(* CODESYS project tc3_linmot_v1_0_0_3_20150204.library
   Company: NTI AG
   Title: Tc3_LinMot
   Author: NTI AG - LinMot
   Version: 1.0.0.3

Project tree, tasks and I/O mapping:
  libraries: Tc2_Standard, 3.3.0.0 (Beckhoff Automation GmbH)
  Data types/
    internal/
      data type tenLM_AxisState
      data type tstLM_DrvToPlc
      data type tstLM_PlcToDrv
    data type tstLM_Axis
    data type tstLM_CfgCTEntry
    data type tstLM_CfgUPIDListEntry
    data type tstLM_CTEntry
    data type tstLM_LiveParameter
  POUs/
    LinMot Axis Control Function Blocks/
      Unofficial_Unsupported/
        function block LMct_AxisCtrlE12x0_Abort [ST]
      function block LMct_AxisControl [ST]
    LinMot CAM Function Blocks/
      function block LMcm_CAMCtrl [ST]
      function block LMcm_LoadCAM1_mc1100 [ST]
      function block LMcm_LoadCAM1_mc1130 [ST]
      function block LMcm_LoadCAM2_mc1200 [ST]
      function block LMcm_LoadCAM2_mc1230 [ST]
    LinMot Config Function Blocks/
      Unofficial_Unsupported/
        function block LMcf_ParaAccessExt [ST]
      function block LMcf_CTAccess [ST]
      function block LMcf_CurveAccess [ST]
      function block LMcf_GetErrorTxt [ST]
      function block LMcf_GetModUPIDList [ST]
      function block LMcf_ParaAccess [ST]
      function block LMcf_StopStartDefault [ST]
      function block LMcf_WriteUPIDList [ST]
    LinMot Force Control Function Blocks/
      Unofficial_Unsupported/
        function block LMfc_ChangeTargetForceCont [ST]
      function block LMfc_ChangeTargetForce [ST]
      function block LMfc_GoToPosForceCtrlHighLim [ST]
      function block LMfc_GoToPosForceCtrlLowLim [ST]
      function block LMfc_GoToPosRstForceCtrl [ST]
    LinMot Functions/
      function F_GetVersionLinMotLibrary [ST]
      function block LM_F_TRIG [ST]
      function block LM_R_TRIG [ST]
      function LM_UptMCI [ST]
      function USINT_TO_ASCIISTRING [ST]
    LinMot MC Function Blocks/
      Unofficial_Unsupported/
        function block LMmt_IncrTargetPos [ST]
      function block LMmt_GenericMC [ST]
      function block LMmt_IncrActPos [ST]
      function block LMmt_MoveAbs [ST]
      function block LMmt_MoveRel [ST]
      function block LMmt_StartCTCommand [ST]
      function block LMmt_Stop [ST]
      function block LMmt_WriteLivePar [ST]
    LinMot MC Function Blocks Advanced/
      Unofficial_Unsupported/
        function block LMav_PVStreamLREAL [ST]
      function block LMav_CurrentCmdMode [ST]
      function block LMav_Mod16BitCTPar [ST]
      function block LMav_Mod32BitCTPar [ST]
      function block LMav_MoveBestehorn [ST]
      function block LMav_MoveSin [ST]
      function block LMav_PStream [ST]
      function block LMav_PVStream [ST]
      function block LMav_RunCurve [ST]
    Rotary Motors/
      function block LMct_RotaryMotorControl [ST]
      function block LMmt_RotIncrActAngle [ST]
      function block LMmt_RotMoveAbs [ST]
      function block LMmt_RotMoveInfNeg [ST]
      function block LMmt_RotMoveInfPos [ST]
      function block LMmt_RotMoveRel [ST]
  Version/
    global variables Global_Version
  Visualizations/
*)

// Data types/internal/tenLM_AxisState
TYPE tenLM_AxisState :
(*PLC Open like naming of the drive state - ! Has no functionality ! *)
(
	Disabled_LM,
	StandStill_LM,
	Homing_LM,
	ErrorStop_LM,
	Stopping_LM,
	DiscreteMotion_LM,
	ContinuousMotion_LM,
	SynchronizedMotion_LM,
	Jogging_LM
);
END_TYPE

// Data types/internal/tstLM_DrvToPlc
TYPE tstLM_DrvToPlc :
STRUCT
	StateVar 			:UINT; (*StateVar of the drive*)
	StatusWord 			:UINT; (*Statusword of the drive*)
	WarnWord 			:UINT; (*Warnword of the drive*)
	ComActualCurrent16 	:INT; (*16Bit actual current For x11x0 series drive*)
	ComDemandPosition 	:DINT; (*32Bit demand position*)
	ComActualPosition 	:DINT; (*32Bit actual position*)
	ComActualCurrent32 	:DINT; (*32Bit actual current For E1200 series drives*)

	CfgStatusWord 		:UINT; (*Config Channel Status*)
	CfgIndexIn 			:UINT; (*Argument (meaning depends on Cmd ID*)
	CfgValueIn 			:UDINT; (*Argument (meaning depends on Cmd ID*)
END_STRUCT
END_TYPE

// Data types/internal/tstLM_PlcToDrv
TYPE tstLM_PlcToDrv :
STRUCT
	ControlWord 		:UINT; (*ControlWord of the drive*)
	MCHeader 			:UINT; (*Motion command header*)
	MCParaWord0 		:UINT; (*Motion command parameter word 0*)
	MCParaWord1 		:UINT; (*Motion command parameter word 1*)
	MCParaWord2 		:UINT; (*Motion command parameter word 2*)
	MCParaWord3 		:UINT; (*Motion command parameter word 3*)
	MCParaWord4 		:UINT; (*Motion command parameter word 4*)
	MCParaWord5 		:UINT; (*Motion command parameter word 5*)
	MCParaWord6 		:UINT; (*Motion command parameter word 6*)
	MCParaWord7 		:UINT; (*Motion command parameter word 7*)
	MCParaWord8 		:UINT; (*Motion command parameter word 8*)
	MCParaWord9 		:UINT; (*Motion command parameter word 9*)
	MCParaWord10 		:UINT; (*Motion command parameter word 10*)
	MCParaWord11 		:UINT; (*Motion command parameter word 11*)
	MCParaWord12 		:UINT; (*Motion command parameter word 12*)
	MCParaWord13 		:UINT; (*Motion command parameter word 13*)
	MCParaDWord_00_03 	:UDINT; (*Motion command parameter bytes 0-3 (used for E12X0 series drives)*)
	MCParaDWord_04_07 	:UDINT; (*Motion command parameter bytes 4-7 (used for E12X0 series drives)*)
	MCParaDWord_08_11 	:UDINT; (*Motion command parameter bytes 8-11 (used for E12X0 series drives)*)
	MCParaDWord_12_15 	:UDINT; (*Motion command parameter bytes 12-15 (used for E12X0 series drives)*)
	MCParaDWord_16_19 	:UDINT; (*Motion command parameter bytes 16-19 (used for E12X0 series drives)*)
	MCParaDWord_20_23 	:UDINT; (*Motion command parameter bytes 20-23 (used for E12X0 series drives)*)
	MCParaDWord_24_27 	:UDINT; (*Motion command parameter bytes 24-27 (used for E12X0 series drives)*)

	CfgControlWord 		:UINT; (*Config Channel Control*)
	CfgIndexOut 		:UINT; (*Argument (meaning depends on Cmd ID*)
	CfgValueOut 		:UDINT; (*Argument (meaning depends on Cmd ID*)
END_STRUCT
END_TYPE

// Data types/tstLM_Axis
TYPE tstLM_Axis : 
STRUCT
	PlcToDrv			AT%Q* :tstLM_PlcToDrv; (*PLC to Drive struct*)
	DrvToPlc			AT%I* :tstLM_DrvToPlc; (*Drive to PLC struct*)
	(*Status information*)
	AxisState			:tenLM_AxisState;
	CommandRunning		:BOOL;
	CommandAborted		:BOOL;
	ConfigChannelBusy	:BOOL;
	(*Information (Not required for prober work of the library function blocks)*)
	AxisName			:STRING;
	AxisNr				:UINT;
	AxisCtrlType		:STRING; (*Eg. 'E1200-EC-UC', 'E1130-DP', 'B1100-GP', ....*)
END_STRUCT
END_TYPE

// Data types/tstLM_CfgCTEntry
TYPE tstLM_CfgCTEntry :
STRUCT
	CTID		:UINT; (*ID of command table entry*)
	BlockSize	:UINT; (*Size of EntryBlock in Bytes*)
	DataBlock	:ARRAY[0..15] OF UDINT; (*EntryBlock, 64Bytes*)

(*Example of a Command Table Entry Data Block:
0002A701h, 	LowWord = Entry Version ID (fix A701h) / HighWord = Sequenced Entry ID
00000100h,	LowWord: Motion Cmd Header(010xh=VAI Go To Pos) / HighWord: Motion Cmd Par Byte 0..1
42400000h, 	Motion Cmd Par Byte 2..5
4240000Fh, 	Motion Cmd Par Byte 6..9
4240000Fh, 	Motion Cmd Par Byte 10..13
0000000Fh, 	Motion Cmd Par Byte 14..17
00000000h, 	Motion Cmd Par Byte 18..21
00000000h, 	Motion Cmd Par Byte 22..25
00000000h, 	Motion Cmd Par Byte 26..29
6E550000h, 	LowWord: Motion Cmd Par Byte 30..31 / HighWord: Entry Name Character 0..1
656D616Eh, 	Entry Name Character 2..5
00000064h, 	Entry Name Character 6..9
00000000h, 	Entry Name Character 10..13
FFFF0000h, 	LowWord: Entry Name Character 14..15 / HighWord: Reserved for future use
FFFFFFFFh, 	Reserved for future use
FFFFFFFFh, 	Reserved for future use
*)
END_STRUCT
END_TYPE

// Data types/tstLM_CfgUPIDListEntry
TYPE tstLM_CfgUPIDListEntry :
STRUCT
	UPID		:UINT; (*LinMot parameter, UPID [Unique Parameter ID]*)
	UPIDValue	:UDINT; (*Value of the parameter*)
END_STRUCT
END_TYPE

// Data types/tstLM_CTEntry
TYPE tstLM_CTEntry :
STRUCT
	CTEntryID	:INT;
	ParaOffset	:INT;
	ParaValue	:DINT;
END_STRUCT
END_TYPE

// Data types/tstLM_LiveParameter
TYPE tstLM_LiveParameter :
STRUCT
	UPID		:UINT;
	UPIDValue	:DINT;
END_STRUCT
END_TYPE

// Version/Global_Version
// This function has been automatically generated from the project information.
VAR_GLOBAL CONSTANT
	{attribute 'const_non_replaced'}
	stLibVersion_Tc3_LinMot : ST_LibVersion := (iMajor := 1, iMinor := 0, iBuild := 0, iRevision := 3, sVersion := '1.0.0.3');
END_VAR

// POUs/LinMot Axis Control Function Blocks/Unofficial_Unsupported/LMct_AxisCtrlE12x0_Abort
FUNCTION_BLOCK LMct_AxisCtrlE12x0_Abort
VAR_INPUT
	SwitchOn			:BOOL;	(*Switch on motor*)
	Abort_INV			:BOOL;	(*/Abort*)
	Home				:BOOL;	(*Start homing procedure*)
	ErrorAcknowledge	:BOOL;	(*Error acknowledge*)
	JogPlus				:BOOL;	(*Jog move postive*)
	JogMinus			:BOOL;	(*Jog move negative*)
END_VAR
VAR_IN_OUT
	Axis				:tstLM_Axis; (*Axis reference*)
END_VAR
VAR_OUTPUT
	OperationEnabled	:BOOL;	(*Axis powered on*)
	Aborting			:BOOL;	(*Aborting*)
	SwitchOnLocked		:BOOL;	(*Switch on locked*)
	Homed				:BOOL;	(*Axis has reference*)
	MotionActive		:BOOL;	(*Motion active (Setpoint generation (VAI, curve) active)*)
	Jogging				:BOOL;	(*Axis is moving in jog mode*)
	Warning				:BOOL;	(*Warning detected*)
	Error				:BOOL; 	(*Error detected*)
	ErrorCode			:UINT;	(*Error code, see MotionCtrlSW manual*)
	ActualPosition		:REAL;	(*Actual position in [mm]*)
	ActualCurrent		:REAL;	(*Actual motor current in [A]*)
END_VAR
VAR
	uiState				:UINT;	(*internal -> Current state of the drive*)
	rTrigHome 			:LM_R_TRIG;	(*internal ->*)
	rTrigHomed 			:LM_R_TRIG;	(*internal ->*)
	bRehome 			:BOOL; 	(*internal ->*)
END_VAR
(*Version history:
Date         	 | Version    	| Created under     		| Author          		| Remark 
------------------------------------------------------------------------------------------------------------------------------- 
2011-jul-12   	 | 1.0.0      	| V2.11.0 (Build 1016)		| fj  					| initial release 
2011-nov-22   	 | 1.0.1      	| V2.11.0 (Build 1016)		| fj  					| homed output reset if home input is set 
2011-dec-01   	 | 1.0.2      	| V2.11.0 (Build 1016)		| fj  					| code optimisation
2012-jan-25   	 | 1.0.3     	| V2.11.0 (Build 1016)		| fj  					| operation enabled output is now directly mapped to the status word bit 0
2012-may-01  	 | 1.1.0b     	| V2.11.0 (Build 1016)		| fj  					| added /Abort input
2012-aug-21  	 | 1.1.0c     	| V2.11.0 (Build 1016)		| fj  					| added additional StateVar check for 090Fh ("homing finished") when rehoming
*)

(*Eingänge zuweisen/lesen ][ Read and allocate inputs*)
	ActualPosition := DINT_TO_REAL(Axis.DrvToPlc.ComActualPosition)/10000;
    	ActualCurrent := DINT_TO_REAL(Axis.DrvToPlc.ComActualCurrent32)/1000;

(*Variablen ][ variables*)
	uiState := SHR(Axis.DrvToPlc.StateVar, 8);
	SwitchOnLocked := Axis.DrvToPlc.StatusWord.6;
	Warning := Axis.DrvToPlc.StatusWord.7;
	Homed := Axis.DrvToPlc.StatusWord.11;
	MotionActive := Axis.DrvToPlc.StatusWord.13;
	OperationEnabled	:= Axis.DrvToPlc.StatusWord.0;

(*	IF uiState = 16#08 THEN
		OperationEnabled	:= Axis.DrvToPlc.StatusWord.0;
	ELSE
		OperationEnabled	:= FALSE;
	END_IF
*) (*Disabled 2012/01/25 fj*)
(*=============================================================================
*  State Machine
===============================================================================*)    

CASE uiState OF
	(*Not Ready to Switch On*)
	00:	Axis.AxisState := Disabled_LM;

	(*State 4: Error*)
	04:	ErrorCode := UINT_TO_USINT(Axis.DrvToPlc.StateVar);
           	Error := TRUE;
		Axis.AxisState := ErrorStop_LM;

	(*State 8: Operation Enabled*)
	08:	Homed := Axis.DrvToPlc.StateVar.7;
		IF Axis.DrvToPlc.StatusWord.13 AND NOT (Axis.AxisState = Stopping_LM) THEN
			Axis.AxisState := DiscreteMotion_LM;
		ELSIF NOT Axis.DrvToPlc.StatusWord.13 AND NOT (Axis.AxisState = Stopping_LM) THEN
			Axis.AxisState := StandStill_LM;
		END_IF

	(*State 9: Homing*)
	09:	Axis.AxisState := Homing_LM;

	(*State 12: Aborting*)
	12:	Aborting := TRUE;
		IF Axis.DrvToPlc.StatusWord.13 THEN
			Axis.AxisState := Stopping_LM;
		ELSE
			Axis.AxisState := StandStill_LM;
		END_IF

	(*State 14: Error Behaviour QuickStop*)
	14:	Axis.AxisState := ErrorStop_LM;

	(*State 16: Jogging +*)
	16:	Axis.AxisState := Jogging_LM;

	(*State 17: Jogging -*)
	17:	Axis.AxisState := Jogging_LM;

END_CASE;


(*Wenn der drive nicht im Fehlerzustand ist, werden Error und ErrorCode auf Null gesetzt*)
(*If the drive is not in Error state, Error and ErrorCode are set to zero*)
IF uiState <> 16#04 THEN
        	Error := FALSE;
        	ErrorCode := 16#00;
END_IF;

IF uiState <> 16#08 THEN
        	Axis.PlcToDrv.MCHeader := 16#0000; (*Reset Header to prevent "MC Cmd in wrong state" error*)
	Axis.CommandRunning := FALSE;
	Axis.CommandAborted := FALSE;
END_IF;

(*Switch On*)
Axis.PlcToDrv.ControlWord.0 := SwitchOn;
IF NOT Axis.PlcToDrv.ControlWord.0 AND NOT (uiState = 4 OR uiState = 12 OR uiState = 14) THEN
	Axis.AxisState := Disabled_LM;
END_IF

(*Home*)
Axis.PlcToDrv.ControlWord.11 := Home;
rTrigHome(CLK:=Home);
rTrigHomed(CLK:=Axis.DrvToPlc.StatusWord.11);

IF rTrigHome.Q AND (uiState = 8) THEN
	bRehome := TRUE;
END_IF
IF bRehome THEN
	Homed := FALSE;
	IF rTrigHomed.Q OR (Axis.DrvToPlc.StateVar = 16#090F) THEN
 		bRehome := FALSE;
  		Homed := Axis.DrvToPlc.StatusWord.11;
	END_IF
END_IF

(*Error acknowledge*)
Axis.PlcToDrv.ControlWord.7 := ErrorAcknowledge;

(*JogPlus*)
Axis.PlcToDrv.ControlWord.8 := JogPlus;

(*JogMinus*)
Axis.PlcToDrv.ControlWord.9 := JogMinus;

IF (uiState = 16 OR uiState = 17) AND UINT_TO_USINT(Axis.DrvToPlc.StateVar) = 16#01 THEN
	Jogging := TRUE;
ELSE
	Jogging := FALSE;
END_IF

(*/Abort*)
Axis.PlcToDrv.ControlWord.4 := Abort_INV;
IF NOT Abort_INV THEN
	Axis.CommandAborted := TRUE;
ELSE
	Aborting := FALSE;
END_IF

END_FUNCTION_BLOCK

// POUs/LinMot Functions/LM_R_TRIG
FUNCTION_BLOCK LM_R_TRIG
(* Rising Edge detection *)
VAR_INPUT
	CLK	:BOOL;	(*Signal to detect*)
END_VAR
VAR_OUTPUT
	Q	:BOOL;	(*Edge detected*)
END_VAR
VAR
	M	:BOOL;
END_VAR
(*Version history:
Date         	 | Version    		| Created under     	| Author          	| Remark 
------------------------------------------------------------------------------------------------------------------------------- 
2013-nov-27   	 | 1.0.0      		| V2.11.0 (Build 1016)	| fj  				| initial release 
*)

(*Bildung der positiven Flanke  // get the positive pulse*)
    Q  := CLK AND NOT M;
    M  := CLK;

END_FUNCTION_BLOCK

// POUs/LinMot Axis Control Function Blocks/LMct_AxisControl
FUNCTION_BLOCK LMct_AxisControl
VAR_INPUT
	SwitchOn		    :BOOL;	(*Switch on motor*)
	Home				:BOOL;	(*Start homing procedure*)
	ErrorAcknowledge	:BOOL;	(*Error acknowledge*)
	JogPlus				:BOOL;	(*Jog move postive*)
	JogMinus			:BOOL;	(*Jog move negative*)
END_VAR
VAR_IN_OUT
	Axis	       		:tstLM_Axis; (*Axis reference*)
END_VAR
VAR_OUTPUT
	OperationEnabled	:BOOL;	(*Axis powered on*)
	SwitchOnLocked		:BOOL;	(*Switch on locked*)
	Homed     	      	:BOOL;	(*Axis has reference*)
	MotionActive		:BOOL;	(*Motion active (Setpoint generation (VAI, curve) active)*)
	Jogging				:BOOL;	(*Axis is moving in jog mode*)
	Warning         	:BOOL;	(*Warning detected*)
	Error          		:BOOL;	(*Error detected*)
	ErrorCode      		:UINT;	(*Error code, see MotionCtrlSW manual*)
	DemandPosition  	:REAL;	(*Demand position in [mm]*)
	ActualPosition  	:REAL;	(*Actual position in [mm]*)
	ActualCurrent   	:REAL;	(*Actual motor current in [A]*)
END_VAR
VAR
	uiState        		:UINT;	(*internal -> Current state of the drive*)
	rTrigHome 			:LM_R_TRIG;	(*internal ->*)
	fTrigHome 			:LM_F_TRIG;	(*internal ->*)
END_VAR
(*Version history:
Date         	 | Version    		| Created under     	| Author          	| Remark 
------------------------------------------------------------------------------------------------------------------------------- 
2011-jul-12   	 | 1.0.0      		| V2.11.0 (Build 1016)	| fj  				| initial release 
2011-nov-22   	 | 1.0.1      		| V2.11.0 (Build 1016)	| fj  				| homed output reset if home input is set 
2011-dec-01   	 | 1.0.2      		| V2.11.0 (Build 1016)	| fj  				| code optimisation
2012-jan-25   	 | 1.0.3     		| V2.11.0 (Build 1016)	| fj  				| operation enabled output is now directly mapped to the status word bit 0
2012-oct-16   	 | 1.1.0      		| V2.11.0 (Build 1016)	| fj  				| added additional StateVar check for 090Fh ("homing finished") when rehoming
2014-may-13   	 | 1.0.0.1     		| v3.14014.0			| fj  				| added output DemandPosition
																				| optimized home input / homed output behaviour
*)

(*Eingänge zuweisen/lesen ][ Read and allocate inputs*)
	ActualPosition := DINT_TO_REAL(Axis.DrvToPlc.ComActualPosition)/10000;
	DemandPosition := DINT_TO_REAL(Axis.DrvToPlc.ComDemandPosition)/10000;
	(*Workaround for different XML current definitions (16Bit/32Bit)*)
	IF Axis.DrvToPlc.ComActualCurrent32 = 0 AND Axis.DrvToPlc.ComActualCurrent16 = 0 THEN
		ActualCurrent := 0;
	ELSIF Axis.DrvToPlc.ComActualCurrent32 <> 0 AND Axis.DrvToPlc.ComActualCurrent16 = 0 THEN
		ActualCurrent := DINT_TO_REAL(Axis.DrvToPlc.ComActualCurrent32)/1000;
	ELSIF Axis.DrvToPlc.ComActualCurrent32 = 0 AND Axis.DrvToPlc.ComActualCurrent16 <> 0 THEN
		ActualCurrent := INT_TO_REAL(Axis.DrvToPlc.ComActualCurrent16)/1000;
	ELSE
		ActualCurrent := DINT_TO_REAL(Axis.DrvToPlc.ComActualCurrent32)/1000; (*If both 16/32Bit currents aren't 0 32Bit has higher priority*)
	END_IF

(*Variablen ][ variables*)
	uiState := SHR(Axis.DrvToPlc.StateVar, 8);
	SwitchOnLocked := Axis.DrvToPlc.StatusWord.6;
	Warning := Axis.DrvToPlc.StatusWord.7;
	MotionActive := Axis.DrvToPlc.StatusWord.13;
	OperationEnabled := Axis.DrvToPlc.StatusWord.0;

(*=============================================================================
*  State Machine
===============================================================================*)    

CASE uiState OF
	(*Not Ready to Switch On*)
	00:	Axis.AxisState := Disabled_LM;

	(*State 4: Error*)
	04:	ErrorCode := UINT_TO_USINT(Axis.DrvToPlc.StateVar);
		Error := TRUE;
		Axis.AxisState := ErrorStop_LM;

	(*State 8: Operation Enabled*)
	08:	Homed := Axis.DrvToPlc.StateVar.7;
		IF Axis.DrvToPlc.StatusWord.13 AND NOT (Axis.AxisState = Stopping_LM) THEN
			Axis.AxisState := DiscreteMotion_LM;
		ELSIF NOT Axis.DrvToPlc.StatusWord.13 AND NOT (Axis.AxisState = Stopping_LM) THEN
			Axis.AxisState := StandStill_LM;
		END_IF

	(*State 9: Homing*)
	09:	Axis.AxisState := Homing_LM;
		IF Axis.DrvToPlc.StateVar = 16#090F THEN
			Axis.PlcToDrv.ControlWord.11 := FALSE;
		END_IF

	(*State 14: Error Behaviour QuickStop*)
	14:	Axis.AxisState := ErrorStop_LM;

	(*State 16: Jogging +*)
	16:	Axis.AxisState := Jogging_LM;

	(*State 17: Jogging -*)
	17:	Axis.AxisState := Jogging_LM;

END_CASE;


(*Wenn der drive nicht im Fehlerzustand ist, werden Error und ErrorCode auf Null gesetzt*)
(*If the drive is not in Error state, Error and ErrorCode are set to zero*)
IF uiState <> 16#04 THEN
	Error := FALSE;
	ErrorCode := 16#00;
END_IF;

IF uiState <> 16#08 THEN
	Axis.PlcToDrv.MCHeader := 16#0000; (*Reset Header to prevent "MC Cmd in wrong state" error*)
	Axis.CommandRunning := FALSE;
	Axis.CommandAborted := FALSE;
END_IF;

(*Switch On*)
Axis.PlcToDrv.ControlWord.0 := SwitchOn;
IF NOT Axis.PlcToDrv.ControlWord.0 AND NOT (uiState = 4 OR uiState = 14) THEN
	Axis.AxisState := Disabled_LM;
END_IF

(*Home*)
rTrigHome(CLK:=Home);
fTrigHome(CLK:=Home);
IF rTrigHome.Q THEN
	Axis.PlcToDrv.ControlWord.11 := TRUE;
END_IF
IF fTrigHome.Q  THEN
	Axis.PlcToDrv.ControlWord.11 := FALSE;
END_IF

IF uiState = 16#09 OR (Axis.PlcToDrv.ControlWord.11 AND NOT (uistate = 16#09)) THEN
	Homed := FALSE;
ELSE
	Homed := Axis.DrvToPlc.StatusWord.11;
END_IF

(*Error acknowledge*)
Axis.PlcToDrv.ControlWord.7 := ErrorAcknowledge;

(*JogPlus*)
Axis.PlcToDrv.ControlWord.8 := JogPlus;

(*JogMinus*)
Axis.PlcToDrv.ControlWord.9 := JogMinus;

IF (uiState = 16 OR uiState = 17) AND UINT_TO_USINT(Axis.DrvToPlc.StateVar) = 16#01 THEN
	Jogging := TRUE;
ELSE
	Jogging := FALSE;
END_IF

END_FUNCTION_BLOCK

// POUs/LinMot Functions/LM_F_TRIG
FUNCTION_BLOCK LM_F_TRIG
(* Falling Edge detection *)
VAR_INPUT
	CLK	:BOOL;	(*Signal to detect*)
END_VAR
VAR_OUTPUT
	Q	:BOOL;	(*Edge detected*)
END_VAR
VAR
	M	:BOOL;
END_VAR
(*Version history:
Date         	 | Version    		| Created under     	| Author          	| Remark 
------------------------------------------------------------------------------------------------------------------------------- 
2013-nov-27   	 | 1.0.0      		| V2.11.0 (Build 1016)	| fj  				| initial release 
*)

(*Bildung der negativen Flanke  // get the negative pulse*)
    Q  := NOT CLK AND M;
    M  := CLK;

END_FUNCTION_BLOCK

// POUs/LinMot CAM Function Blocks/LMcm_CAMCtrl
FUNCTION_BLOCK LMcm_CAMCtrl
VAR_INPUT
	Execute			:BOOL;	(*Execute command*)
	Mode			:UINT;	(*Mode 0: CAM Enable
 							Mode 1: CAM Disable
 							Mode 2: CAM Go To Sync Pos
 							Mode 3: Encoder CAM Set Value [Inputs used: EncValue]
							Mode 4: Encoder CAM 1 Enable
							Mode 5: Encoder CAM 1 Disable
							Mode 6: Encoder CAM 2 Enable
							Mode 7: Encoder CAM 2 Disable
							*)
	EncValue		:UDINT;	(*Encoder value to be written*)
END_VAR
VAR_IN_OUT
	Axis	        			:tstLM_Axis; (*Axis reference*)
END_VAR
VAR_OUTPUT
	Done			:BOOL;	(*Command has been executed*)
	Busy			:BOOL;	(*Command running / FB Busy*)
	Error          	:BOOL;	(*Error detected*)
	ErrorID 		:UINT;	(*Error ID:
							01h: Axis not ready
 							02h: Axis already has command running
 							03h: Axis has error
 							04h: Command interrupted
 							05h: Command aborted
							06h: Invalid input(s)
							*)
END_VAR
VAR
	usiOldCmdCount 	:USINT;	(*internal -> *)
	usiNewCmdCount	:USINT; 	(*internal -> *)
	uiCState		:UINT;     	(*internal -> *)
	uiFbState		:UINT;	(*internal -> *)
	rTrig			:LM_R_TRIG;	(*internal -> *)
	uiCmdHeader		:UINT;	(*internal -> *)
END_VAR

(*Version history:
Date         	 | Version    		| Created under     	| Author       		| Remark 
------------------------------------------------------------------------------------------------------------------------------- 
2012-aug-30   	 | 1.1.0     		| V2.11.0 (Build 1016)	| fj  				| initial release
2013-nov-27   	 | 1.1.1      		| V2.11.0 (Build 1016)	| fj  				| check if command done fixed
*)

	usiOldCmdCount := SHR(UINT_TO_USINT(SHL(Axis.DrvToPlc.StateVar,4)),4);
	uiCState := SHR(Axis.DrvToPlc.StateVar, 8);

(*Flankenerkennung am Execute Eingang*)
(*Edge detection on Execute input*)
rTrig(CLK:=Execute);
IF rTrig.Q AND Mode = 2 AND uiCState = 16#08 AND Axis.DrvToPlc.StateVar.6 AND NOT Axis.CommandRunning THEN (*Start command if mode = 2*)
	Axis.CommandRunning := TRUE;
	Busy := TRUE;
	uiFbState := 1;
ELSIF rTrig.Q AND Mode <> 2 AND NOT  Axis.CommandRunning THEN (*Start command if mode <> 2*)
	Axis.CommandRunning := TRUE;
	Busy := TRUE;
	uiFbState := 1;
ELSIF rTrig.Q AND Mode = 2 AND (uiCState <> 16#08 OR NOT Axis.DrvToPlc.StateVar.6) THEN (*Axis not ready*)
	uiFbState := 50; (*Error state*)
	Error := TRUE;
	ErrorID := 16#01; (*Axis not ready*)
ELSIF rTrig.Q AND Axis.CommandRunning AND NOT Busy THEN (*Axis already has a command running*)
	uiFbState := 50; (*Error state*)
	Error := TRUE;
	ErrorID := 16#02; (*Axis already has a command running*)
END_IF

IF Busy AND Mode = 2 AND uiCState = 16#04 THEN
	Axis.CommandRunning := FALSE;
	uiFbState := 50;
	Error := TRUE;
	ErrorID := 16#03; (*Axis has error*)
END_IF

IF Busy AND Mode = 2 AND uiCState <> 16#08 THEN
	Axis.CommandRunning := FALSE;
	uiFbState := 50; (*Error state*)
	Error := TRUE;
	ErrorID := 16#04; (*Command interupted*)
ELSIF Busy AND Axis.CommandAborted THEN
	uiFbState := 50; (*Error state*)
	Error := TRUE;
	ErrorID := 16#05; (*Command aborted*)
END_IF

(*State machine*)
CASE uiFbState OF
	0:	;

	1:     	(*Befehlskopf mit CMD Count berechen und senden ][ Calculate and send command header*)
		CASE Mode OF
			0:	uiCmdHeader := 16#1000; (*CAM Enable*)
			1:	uiCmdHeader := 16#1010; (*CAM Disable*)
			2:	uiCmdHeader := 16#1020; (*CAM Go To Sync Pos*)
			3:	uiCmdHeader := 16#1040; (*Encoder CAM Set Value*)
			4:	uiCmdHeader := 16#1160; (*Encoder CAM 1 Enable*)
			5:	uiCmdHeader := 16#1170; (*Encoder CAM 1 Disable*)
			6:	uiCmdHeader := 16#1260; (*Encoder CAM 2 Enable*)
			7:	uiCmdHeader := 16#1270; (*Encoder CAM 2 Disable*)
		END_CASE

		usiNewCmdCount := (usiOldCmdCount + 1) MOD 16 ; (*MOD 16*)
     	   	Axis.PlcToDrv.MCHeader := 16#0000; (*Reset Header*)
     	   	Axis.PlcToDrv.MCHeader := uiCmdHeader + usiNewCmdCount;

		IF Mode = 3 THEN
			Axis.PlcToDrv.MCParaWord0 := UDINT_TO_UINT(EncValue);
			Axis.PlcToDrv.MCParaWord1 := UDINT_TO_UINT(ROR(EncValue,16));
		ELSE
			Axis.PlcToDrv.MCParaWord0 := 0;
			Axis.PlcToDrv.MCParaWord1 := 0;
		END_IF

		LM_UptMCI(Axis);

		uiFbState := 2;

	2:	(*Prüfen ob Befehl ausgeführt ][ Check if command has been executed*)
		IF (Mode = 2 AND (usiOldCmdCount = usiNewCmdCount) AND uiCState = 16#08 AND Axis.DrvToPlc.StateVar.6)
			OR ((Mode <> 2) AND (usiOldCmdCount = usiNewCmdCount)) THEN
			Done := TRUE;
			Busy := FALSE;
	     	   	Axis.PlcToDrv.MCHeader := 16#0000 + usiNewCmdCount; (*Send no operation*)
			Axis.CommandRunning := FALSE;
			uiFbState := 3;
		END_IF

	3:	IF NOT Execute THEN
			uiFbState := 0;
			Busy := FALSE;
			Done := FALSE;
		END_IF

	50:	Error := TRUE;
		Busy := FALSE;
		Done := FALSE;
		IF NOT Execute THEN
			uiFbState := 0;
			Error := FALSE;
			ErrorID := 0;
		END_IF

END_CASE

END_FUNCTION_BLOCK

// POUs/LinMot Functions/LM_UptMCI
FUNCTION LM_UptMCI : bool
VAR_IN_OUT
	Axis 	:tstLM_Axis;
END_VAR
VAR
END_VAR

Axis.PlcToDrv.MCParaDWord_00_03 := SHL(UINT_TO_UDINT(Axis.PlcToDrv.MCParaWord1),16) + UINT_TO_UDINT(Axis.PlcToDrv.MCParaWord0);
Axis.PlcToDrv.MCParaDWord_04_07 := SHL(UINT_TO_UDINT(Axis.PlcToDrv.MCParaWord3),16) + UINT_TO_UDINT(Axis.PlcToDrv.MCParaWord2);
Axis.PlcToDrv.MCParaDWord_08_11 := SHL(UINT_TO_UDINT(Axis.PlcToDrv.MCParaWord5),16) + UINT_TO_UDINT(Axis.PlcToDrv.MCParaWord4);
Axis.PlcToDrv.MCParaDWord_12_15 := SHL(UINT_TO_UDINT(Axis.PlcToDrv.MCParaWord7),16) + UINT_TO_UDINT(Axis.PlcToDrv.MCParaWord6);
Axis.PlcToDrv.MCParaDWord_16_19 := SHL(UINT_TO_UDINT(Axis.PlcToDrv.MCParaWord9),16) + UINT_TO_UDINT(Axis.PlcToDrv.MCParaWord8);
Axis.PlcToDrv.MCParaDWord_20_23 := SHL(UINT_TO_UDINT(Axis.PlcToDrv.MCParaWord11),16) + UINT_TO_UDINT(Axis.PlcToDrv.MCParaWord10);
Axis.PlcToDrv.MCParaDWord_24_27 := SHL(UINT_TO_UDINT(Axis.PlcToDrv.MCParaWord13),16) + UINT_TO_UDINT(Axis.PlcToDrv.MCParaWord12);

END_FUNCTION

// POUs/LinMot CAM Function Blocks/LMcm_LoadCAM1_mc1100
FUNCTION_BLOCK LMcm_LoadCAM1_mc1100
VAR_INPUT
	Execute			:BOOL;    	(*Execute Command*)
	CurveID			:UINT;     	(*Curve ID*)
	CurveStartCount	:UDINT;	(*Curve Start Count [Incr]*)
END_VAR
VAR_IN_OUT
	Axis			:tstLM_Axis; (*Axis struct*)
END_VAR
VAR_OUTPUT
	Done			:BOOL;	(*Command has been executed*)
	Busy			:BOOL;	(*Command running / FB Busy*)
	Error			:BOOL;	(*Error detected*)
	ErrorID			:UINT;	(*Error ID:
							01h: Axis not ready
 							02h: Axis already has command running
 							03h: Axis has error
 							04h: Command interrupted
 							05h: Command aborted
							06h: Invalid input(s)
							*)
END_VAR
VAR
	usiOldCmdCount 	:USINT;	(*internal -> *)
	usiNewCmdCount	:USINT;	(*internal -> *)
	uiCState		:UINT;	(*internal -> *)
	uiFbState		:UINT;	(*internal -> *)
	rTrig			:LM_R_TRIG;	(*internal -> *)
	udiTmpDWord		:UDINT;	(*internal -> *)

 	uiCmdHeader 	:UINT := 16#1100;	(*CommandHeader (110xh) of the "Encoder CAM 1 Define Curve With Default Parameters (110xh)" motion command*)
END_VAR
(*Version history:
Date         	 | Version    	| Created under     		| Author          		| Remark 
------------------------------------------------------------------------------------------------------------------------------- 
2012-aug-30   	 | 1.1.0     		| V2.11.0 (Build 1016)	| fj  				| initial release
*)

(*Variablen ][ variables*)
	usiOldCmdCount := SHR(UINT_TO_USINT(SHL(Axis.DrvToPlc.StateVar,4)),4);
	uiCState := SHR(Axis.DrvToPlc.StateVar, 8);

(*Flankenerkennung am Execute Eingang*)
(*Edge detection on Execute input*)
rTrig(CLK:=Execute);
IF rTrig.Q AND uiCState = 16#08 AND NOT Axis.CommandRunning THEN (*Start command*)
	Axis.CommandRunning := TRUE;
	Busy := TRUE;
	uiFbState := 1;
ELSIF rTrig.Q AND Busy THEN (*Restart command / New rising edge on execute input*)
	Axis.CommandRunning := TRUE;
	Busy := TRUE;
	uiFbState := 1;
ELSIF rTrig.Q AND uiCState <> 16#08 THEN (*Axis not ready*)
	uiFbState := 50; (*Error state*)
	Error := TRUE;
	ErrorID := 16#01; (*Axis not ready*)
ELSIF rTrig.Q AND Axis.CommandRunning AND NOT Busy THEN (*Axis already has a command running*)
	uiFbState := 50; (*Error state*)
	Error := TRUE;
	ErrorID := 16#02; (*Axis already has a command running*)
END_IF

IF Busy AND uiCState = 16#04 THEN
	Axis.CommandRunning := FALSE;
	uiFbState := 50;
	Error := TRUE;
	ErrorID := 16#03; (*Axis has error*)
END_IF

IF Busy AND uiCState <> 16#08 THEN
	Axis.CommandRunning := FALSE;
	uiFbState := 50; (*Error state*)
	Error := TRUE;
	ErrorID := 16#04; (*Command interupted*)
ELSIF Busy AND Axis.CommandAborted THEN
	uiFbState := 50; (*Error state*)
	Error := TRUE;
	ErrorID := 16#05; (*Command aborted*)
END_IF

(*State machine*)
CASE uiFbState OF
	0:	;

	1:	IF (1 <= CurveID AND CurveID <= 100)
		AND (0 <= CurveStartCount AND CurveStartCount <= 4294967295)
		THEN
			(*Befehlskopf mit CMD Count berechen und senden ][ Calculate and send command header*)
			usiNewCmdCount := (usiOldCmdCount + 1) MOD 16 ; (*MOD 16*)
			Axis.PlcToDrv.MCHeader := 16#0000; (*Reset Header*)
			Axis.PlcToDrv.MCHeader := uiCmdHeader + usiNewCmdCount;
	
			Axis.PlcToDrv.MCParaWord0 := CurveID; (*Curve ID*)
	
			Axis.PlcToDrv.MCParaWord1 := UDINT_TO_UINT(CurveStartCount); (*Curve Start Count*)
			Axis.PlcToDrv.MCParaWord2 := UDINT_TO_UINT(ROR(CurveStartCount,16));

			LM_UptMCI(Axis);

			uiFbState := 2;
		ELSE
			Axis.CommandRunning := FALSE;
			uiFbState := 50; (*Error state*)
			Error := TRUE;
			ErrorID := 16#06; (*Invalid input(s)*)
		END_IF

	2:	(*Prüfen ob Befehl ausgeführt ][ Check if command has been executed*)
		IF usiOldCmdCount = usiNewCmdCount AND uiCState = 16#08 THEN
			Done := TRUE;
			Busy := FALSE;
			Axis.PlcToDrv.MCHeader := 16#0000 + usiNewCmdCount; (*Send no operation*)
			Axis.CommandRunning := FALSE;
			uiFbState := 3;
		END_IF

	3:	IF NOT Execute THEN
			uiFbState := 0;
			Busy := FALSE;
			Done := FALSE;
		END_IF

	50:	Error := TRUE;
		Busy := FALSE;
		Done := FALSE;
		IF NOT Execute THEN
			uiFbState := 0;
			Error := FALSE;
			ErrorID := 0;
		END_IF

END_CASE

END_FUNCTION_BLOCK

// POUs/LinMot CAM Function Blocks/LMcm_LoadCAM1_mc1130
FUNCTION_BLOCK LMcm_LoadCAM1_mc1130
VAR_INPUT
	Execute			:BOOL;	(*Execute Command*)
	CurveID			:UINT;	(*Curve ID*)
	CurveStartCount	:UDINT;	(*Curve Start Count [Incr]*)
	OffsetPosition	:REAL;	(*Offset Position [mm]*)
	TargetPosition	:REAL;	(*Target Positon [mm]*)
	CurveLength		:UDINT;	(*Curve Length [Incr]*)
END_VAR
VAR_IN_OUT
	Axis			:tstLM_Axis; (*Axis struct*)
END_VAR
VAR_OUTPUT
	Done			:BOOL;	(*Command has been executed*)
	Busy			:BOOL;	(*Command running / FB Busy*)
	Error			:BOOL;	(*Error detected*)
	ErrorID			:UINT;	(*Error ID:
							01h: Axis not ready
 							02h: Axis already has command running
 							03h: Axis has error
 							04h: Command interrupted
 							05h: Command aborted
							06h: Invalid input(s)
							*)
END_VAR
VAR
	usiOldCmdCount 	:USINT;	(*internal -> *)
	usiNewCmdCount	:USINT;	(*internal -> *)
	uiCState		:UINT;	(*internal -> *)
	uiFbState		:UINT;	(*internal -> *)
	rTrig			:LM_R_TRIG;	(*internal -> *)
	udiTmpDWord		:UDINT;	(*internal -> *)

 	uiCmdHeader 	:UINT := 16#1130;	(*CommandHeader (113xh) of the "Encoder CAM 1 Define Curve From Pos To Pos In Counts (113xh)" motion command*)
END_VAR
(*Version history:
Date         	 | Version    	| Created under     		| Author          		| Remark 
------------------------------------------------------------------------------------------------------------------------------- 
2011-jul-12   	 | 1.0.0      		| V2.11.0 (Build 1016)	| fj  				| initial release 
2011-dec-01   	 | 1.0.2      		| V2.11.0 (Build 1016)	| fj  				| code optimisation
2012-apr-25   	 | 1.1.0     		| V2.11.0 (Build 1016)	| fj  				| added input parameters check
*)

(*Variablen ][ variables*)
	usiOldCmdCount := SHR(UINT_TO_USINT(SHL(Axis.DrvToPlc.StateVar,4)),4);
	uiCState := SHR(Axis.DrvToPlc.StateVar, 8);

(*Flankenerkennung am Execute Eingang*)
(*Edge detection on Execute input*)
rTrig(CLK:=Execute);
IF rTrig.Q AND uiCState = 16#08 AND NOT Axis.CommandRunning THEN (*Start command*)
	Axis.CommandRunning := TRUE;
	Busy := TRUE;
	uiFbState := 1;
ELSIF rTrig.Q AND Busy THEN (*Restart command / New rising edge on execute input*)
	Axis.CommandRunning := TRUE;
	Busy := TRUE;
	uiFbState := 1;
ELSIF rTrig.Q AND uiCState <> 16#08 THEN (*Axis not ready*)
	uiFbState := 50; (*Error state*)
	Error := TRUE;
	ErrorID := 16#01; (*Axis not ready*)
ELSIF rTrig.Q AND Axis.CommandRunning AND NOT Busy THEN (*Axis already has a command running*)
	uiFbState := 50; (*Error state*)
	Error := TRUE;
	ErrorID := 16#02; (*Axis already has a command running*)
END_IF

IF Busy AND uiCState = 16#04 THEN
	Axis.CommandRunning := FALSE;
	uiFbState := 50;
	Error := TRUE;
	ErrorID := 16#03; (*Axis has error*)
END_IF

IF Busy AND uiCState <> 16#08 THEN
	Axis.CommandRunning := FALSE;
	uiFbState := 50; (*Error state*)
	Error := TRUE;
	ErrorID := 16#04; (*Command interupted*)
ELSIF Busy AND Axis.CommandAborted THEN
	uiFbState := 50; (*Error state*)
	Error := TRUE;
	ErrorID := 16#05; (*Command aborted*)
END_IF

(*State machine*)
CASE uiFbState OF
	0:	;

	1:	IF (1 <= CurveID AND CurveID <= 100)
		AND (0 <= CurveStartCount AND CurveStartCount <= 4294967295)
		AND (-214748.0 <= OffsetPosition AND OffsetPosition <= 214748.0)
		AND (-214748.0 <=  TargetPosition AND TargetPosition <= 214748.0)
		AND (0 < CurveLength AND CurveLength <= 4294967295)
		THEN
			(*Befehlskopf mit CMD Count berechen und senden ][ Calculate and send command header*)
			usiNewCmdCount := (usiOldCmdCount + 1) MOD 16 ; (*MOD 16*)
			Axis.PlcToDrv.MCHeader := 16#0000; (*Reset Header*)
			Axis.PlcToDrv.MCHeader := uiCmdHeader + usiNewCmdCount;
	
			Axis.PlcToDrv.MCParaWord0 := CurveID; (*Curve ID*)
	
			Axis.PlcToDrv.MCParaWord1 := UDINT_TO_UINT(CurveStartCount); (*Curve Start Count*)
			Axis.PlcToDrv.MCParaWord2 := UDINT_TO_UINT(ROR(CurveStartCount,16));
	
			udiTmpDWord := DINT_TO_UDINT(REAL_TO_DINT(OffsetPosition * 10000)); (*Offset Position*)
			Axis.PlcToDrv.MCParaWord3 := UDINT_TO_UINT(udiTmpDWord);
			Axis.PlcToDrv.MCParaWord4 := UDINT_TO_UINT(ROR(udiTmpDWord,16));
	
			udiTmpDWord := DINT_TO_UDINT(REAL_TO_DINT(TargetPosition * 10000)); (*Target Position*)
			Axis.PlcToDrv.MCParaWord5 := UDINT_TO_UINT(udiTmpDWord);
			Axis.PlcToDrv.MCParaWord6 := UDINT_TO_UINT(ROR(udiTmpDWord,16));
	
			Axis.PlcToDrv.MCParaWord7 := UDINT_TO_UINT(CurveLength); (*Curve Length*)
			Axis.PlcToDrv.MCParaWord8 := UDINT_TO_UINT(ROR(CurveLength,16));

			LM_UptMCI(Axis);

			uiFbState := 2;
		ELSE
			Axis.CommandRunning := FALSE;
			uiFbState := 50; (*Error state*)
			Error := TRUE;
			ErrorID := 16#06; (*Invalid input(s)*)
		END_IF

	2:	(*Prüfen ob Befehl ausgeführt ][ Check if command has been executed*)
		IF usiOldCmdCount = usiNewCmdCount AND uiCState = 16#08 THEN
			Done := TRUE;
			Busy := FALSE;
			Axis.PlcToDrv.MCHeader := 16#0000 + usiNewCmdCount; (*Send no operation*)
			Axis.CommandRunning := FALSE;
			uiFbState := 3;
		END_IF

	3:	IF NOT Execute THEN
			uiFbState := 0;
			Busy := FALSE;
			Done := FALSE;
		END_IF

	50:	Error := TRUE;
		Busy := FALSE;
		Done := FALSE;
		IF NOT Execute THEN
			uiFbState := 0;
			Error := FALSE;
			ErrorID := 0;
		END_IF

END_CASE;

END_FUNCTION_BLOCK

// POUs/LinMot CAM Function Blocks/LMcm_LoadCAM2_mc1200
FUNCTION_BLOCK LMcm_LoadCAM2_mc1200
VAR_INPUT
	Execute			:BOOL;	(*Execute Command*)
	CurveID			:UINT;	(*Curve ID*)
	CurveStartCount	:UDINT;	(*Curve Start Count [Incr]*)
	OffsetPosition	:REAL;	(*Offset Position [mm]*)
	TargetPosition	:REAL;	(*Target Positon [mm]*)
	CurveLength		:UDINT;	(*Curve Length [Incr]*)
END_VAR
VAR_IN_OUT
	Axis			:tstLM_Axis; (*Axis struct*)
END_VAR
VAR_OUTPUT
	Done			:BOOL;	(*Command has been executed*)
	Busy			:BOOL;	(*Command running / FB Busy*)
	Error			:BOOL;	(*Error detected*)
	ErrorID			:UINT;	(*Error ID:
							01h: Axis not ready
 							02h: Axis already has command running
 							03h: Axis has error
 							04h: Command interrupted
 							05h: Command aborted
							06h: Invalid input(s)
							*)
END_VAR
VAR
	usiOldCmdCount 	:USINT;	(*internal -> *)
	usiNewCmdCount	:USINT;	(*internal -> *)
	uiCState		:UINT;	(*internal -> *)
	uiFbState		:UINT;	(*internal -> *)
	rTrig			:LM_R_TRIG;	(*internal -> *)
	udiTmpDWord		:UDINT;	(*internal -> *)

 	uiCmdHeader 	:UINT := 16#1200;	(*CommandHeader (123xh) of the "Encoder CAM 2 Define Curve With Default Parameters (120xh)" motion command*)
END_VAR
(*Version history:
Date         	 | Version    	| Created under     		| Author          		| Remark 
------------------------------------------------------------------------------------------------------------------------------- 
2012-aug-30   	 | 1.1.0     		| V2.11.0 (Build 1016)	| fj  				| initial release
*)

(*Variablen ][ variables*)
	usiOldCmdCount := SHR(UINT_TO_USINT(SHL(Axis.DrvToPlc.StateVar,4)),4);
	uiCState := SHR(Axis.DrvToPlc.StateVar, 8);

(*Flankenerkennung am Execute Eingang*)
(*Edge detection on Execute input*)
rTrig(CLK:=Execute);
IF rTrig.Q AND uiCState = 16#08 AND NOT Axis.CommandRunning THEN (*Start command*)
	Axis.CommandRunning := TRUE;
	Busy := TRUE;
	uiFbState := 1;
ELSIF rTrig.Q AND Busy THEN (*Restart command / New rising edge on execute input*)
	Axis.CommandRunning := TRUE;
	Busy := TRUE;
	uiFbState := 1;
ELSIF rTrig.Q AND uiCState <> 16#08 THEN (*Axis not ready*)
	uiFbState := 50; (*Error state*)
	Error := TRUE;
	ErrorID := 16#01; (*Axis not ready*)
ELSIF rTrig.Q AND Axis.CommandRunning AND NOT Busy THEN (*Axis already has a command running*)
	uiFbState := 50; (*Error state*)
	Error := TRUE;
	ErrorID := 16#02; (*Axis already has a command running*)
END_IF

IF Busy AND uiCState = 16#04 THEN
	Axis.CommandRunning := FALSE;
	uiFbState := 50;
	Error := TRUE;
	ErrorID := 16#03; (*Axis has error*)
END_IF

IF Busy AND uiCState <> 16#08 THEN
	Axis.CommandRunning := FALSE;
	uiFbState := 50; (*Error state*)
	Error := TRUE;
	ErrorID := 16#04; (*Command interupted*)
ELSIF Busy AND Axis.CommandAborted THEN
	uiFbState := 50; (*Error state*)
	Error := TRUE;
	ErrorID := 16#05; (*Command aborted*)
END_IF

(*State machine*)
CASE uiFbState OF
	0:	;

	1:	IF (1 <= CurveID AND CurveID <= 100)
		AND (0 <= CurveStartCount AND CurveStartCount <= 4294967295)
		THEN
			(*Befehlskopf mit CMD Count berechen und senden ][ Calculate and send command header*)
			usiNewCmdCount := (usiOldCmdCount + 1) MOD 16 ; (*MOD 16*)
			Axis.PlcToDrv.MCHeader := 16#0000; (*Reset Header*)
			Axis.PlcToDrv.MCHeader := uiCmdHeader + usiNewCmdCount;
	
			Axis.PlcToDrv.MCParaWord0 := CurveID; (*Curve ID*)
	
			Axis.PlcToDrv.MCParaWord1 := UDINT_TO_UINT(CurveStartCount); (*Curve Start Count*)
			Axis.PlcToDrv.MCParaWord2 := UDINT_TO_UINT(ROR(CurveStartCount,16));

			LM_UptMCI(Axis);

			uiFbState := 2;
		ELSE
			Axis.CommandRunning := FALSE;
			uiFbState := 50; (*Error state*)
			Error := TRUE;
			ErrorID := 16#06; (*Invalid input(s)*)
		END_IF

	2:	(*Prüfen ob Befehl ausgeführt ][ Check if command has been executed*)
		IF usiOldCmdCount = usiNewCmdCount AND uiCState = 16#08 THEN
			Done := TRUE;
			Busy := FALSE;
			Axis.PlcToDrv.MCHeader := 16#0000 + usiNewCmdCount; (*Send no operation*)
			Axis.CommandRunning := FALSE;
			uiFbState := 3;
		END_IF

	3:	IF NOT Execute THEN
			uiFbState := 0;
			Busy := FALSE;
			Done := FALSE;
		END_IF

	50:	Error := TRUE;
		Busy := FALSE;
		Done := FALSE;
		IF NOT Execute THEN
			uiFbState := 0;
			Error := FALSE;
			ErrorID := 0;
		END_IF

END_CASE

END_FUNCTION_BLOCK

// POUs/LinMot CAM Function Blocks/LMcm_LoadCAM2_mc1230
FUNCTION_BLOCK LMcm_LoadCAM2_mc1230
VAR_INPUT
	Execute			:BOOL;	(*Execute Command*)
	CurveID			:UINT;	(*Curve ID*)
	CurveStartCount	:UDINT;	(*Curve Start Count [Incr]*)
	OffsetPosition	:REAL;	(*Offset Position [mm]*)
	TargetPosition	:REAL;	(*Target Positon [mm]*)
	CurveLength		:UDINT;	(*Curve Length [Incr]*)
END_VAR
VAR_IN_OUT
	Axis			:tstLM_Axis; (*Axis struct*)
END_VAR
VAR_OUTPUT
	Done			:BOOL;	(*Command has been executed*)
	Busy			:BOOL;	(*Command running / FB Busy*)
	Error			:BOOL;	(*Error detected*)
	ErrorID			:UINT;	(*Error ID:
							01h: Axis not ready
 							02h: Axis already has command running
 							03h: Axis has error
 							04h: Command interrupted
 							05h: Command aborted
							06h: Invalid input(s)
							*)
END_VAR
VAR
	usiOldCmdCount 	:USINT;	(*internal -> *)
	usiNewCmdCount	:USINT;	(*internal -> *)
	uiCState		:UINT;	(*internal -> *)
	uiFbState		:UINT;	(*internal -> *)
	rTrig			:LM_R_TRIG;	(*internal -> *)
	udiTmpDWord		:UDINT;	(*internal -> *)

 	uiCmdHeader 	:UINT := 16#1230;	(*CommandHeader (123xh) of the "Encoder CAM 2 Define Curve From Pos To Pos In Counts (113xh)" motion command*)
END_VAR
(*Version history:
Date         	 | Version    	| Created under     		| Author          		| Remark 
------------------------------------------------------------------------------------------------------------------------------- 
2012-aug-30   	 | 1.1.0     		| V2.11.0 (Build 1016)	| fj  				| initial release
*)

(*Variablen ][ variables*)
	usiOldCmdCount := SHR(UINT_TO_USINT(SHL(Axis.DrvToPlc.StateVar,4)),4);
	uiCState := SHR(Axis.DrvToPlc.StateVar, 8);

(*Flankenerkennung am Execute Eingang*)
(*Edge detection on Execute input*)
rTrig(CLK:=Execute);
IF rTrig.Q AND uiCState = 16#08 AND NOT Axis.CommandRunning THEN (*Start command*)
	Axis.CommandRunning := TRUE;
	Busy := TRUE;
	uiFbState := 1;
ELSIF rTrig.Q AND Busy THEN (*Restart command / New rising edge on execute input*)
	Axis.CommandRunning := TRUE;
	Busy := TRUE;
	uiFbState := 1;
ELSIF rTrig.Q AND uiCState <> 16#08 THEN (*Axis not ready*)
	uiFbState := 50; (*Error state*)
	Error := TRUE;
	ErrorID := 16#01; (*Axis not ready*)
ELSIF rTrig.Q AND Axis.CommandRunning AND NOT Busy THEN (*Axis already has a command running*)
	uiFbState := 50; (*Error state*)
	Error := TRUE;
	ErrorID := 16#02; (*Axis already has a command running*)
END_IF

IF Busy AND uiCState = 16#04 THEN
	Axis.CommandRunning := FALSE;
	uiFbState := 50;
	Error := TRUE;
	ErrorID := 16#03; (*Axis has error*)
END_IF

IF Busy AND uiCState <> 16#08 THEN
	Axis.CommandRunning := FALSE;
	uiFbState := 50; (*Error state*)
	Error := TRUE;
	ErrorID := 16#04; (*Command interupted*)
ELSIF Busy AND Axis.CommandAborted THEN
	uiFbState := 50; (*Error state*)
	Error := TRUE;
	ErrorID := 16#05; (*Command aborted*)
END_IF

(*State machine*)
CASE uiFbState OF
	0:	;

	1:	IF (1 <= CurveID AND CurveID <= 100)
		AND (0 <= CurveStartCount AND CurveStartCount <= 4294967295)
		AND (-214748.0 <= OffsetPosition AND OffsetPosition <= 214748.0)
		AND (-214748.0 <=  TargetPosition AND TargetPosition <= 214748.0)
		AND (0 < CurveLength AND CurveLength <= 4294967295)
		THEN
			(*Befehlskopf mit CMD Count berechen und senden ][ Calculate and send command header*)
			usiNewCmdCount := (usiOldCmdCount + 1) MOD 16 ; (*MOD 16*)
			Axis.PlcToDrv.MCHeader := 16#0000; (*Reset Header*)
			Axis.PlcToDrv.MCHeader := uiCmdHeader + usiNewCmdCount;
	
			Axis.PlcToDrv.MCParaWord0 := CurveID; (*Curve ID*)
	
			Axis.PlcToDrv.MCParaWord1 := UDINT_TO_UINT(CurveStartCount); (*Curve Start Count*)
			Axis.PlcToDrv.MCParaWord2 := UDINT_TO_UINT(ROR(CurveStartCount,16));
	
			udiTmpDWord := DINT_TO_UDINT(REAL_TO_DINT(OffsetPosition * 10000)); (*Offset Position*)
			Axis.PlcToDrv.MCParaWord3 := UDINT_TO_UINT(udiTmpDWord);
			Axis.PlcToDrv.MCParaWord4 := UDINT_TO_UINT(ROR(udiTmpDWord,16));
	
			udiTmpDWord := DINT_TO_UDINT(REAL_TO_DINT(TargetPosition * 10000)); (*Target Position*)
			Axis.PlcToDrv.MCParaWord5 := UDINT_TO_UINT(udiTmpDWord);
			Axis.PlcToDrv.MCParaWord6 := UDINT_TO_UINT(ROR(udiTmpDWord,16));
	
			Axis.PlcToDrv.MCParaWord7 := UDINT_TO_UINT(CurveLength); (*Curve Length*)
			Axis.PlcToDrv.MCParaWord8 := UDINT_TO_UINT(ROR(CurveLength,16));

			LM_UptMCI(Axis);

			uiFbState := 2;
		ELSE
			Axis.CommandRunning := FALSE;
			uiFbState := 50; (*Error state*)
			Error := TRUE;
			ErrorID := 16#06; (*Invalid input(s)*)
		END_IF

	2:	(*Prüfen ob Befehl ausgeführt ][ Check if command has been executed*)
		IF usiOldCmdCount = usiNewCmdCount AND uiCState = 16#08 THEN
			Done := TRUE;
			Busy := FALSE;
			Axis.PlcToDrv.MCHeader := 16#0000 + usiNewCmdCount; (*Send no operation*)
			Axis.CommandRunning := FALSE;
			uiFbState := 3;
		END_IF

	3:	IF NOT Execute THEN
			uiFbState := 0;
			Busy := FALSE;
			Done := FALSE;
		END_IF

	50:	Error := TRUE;
		Busy := FALSE;
		Done := FALSE;
		IF NOT Execute THEN
			uiFbState := 0;
			Error := FALSE;
			ErrorID := 0;
		END_IF

END_CASE

END_FUNCTION_BLOCK

// POUs/LinMot Config Function Blocks/Unofficial_Unsupported/LMcf_ParaAccessExt
FUNCTION_BLOCK LMcf_ParaAccessExt
VAR_INPUT
	Execute			:BOOL;	(*Execute command*)
	Mode			:UINT;	(*Mode 0: Read ROM Value of Parameter by UPID [Inputs used: UPIDIn]
 							Mode 1: Read RAM Value of Parameter by UPID [Inputs used: UPIDIn]
 							Mode 2: Write ROM Value of Parameter by UPID [Inputs used: UPIDIn, ValueIn]
 							Mode 3: Write RAM Value of Parameter by UPID [Inputs used: UPIDIn, ValueIn]
 							Mode 4: Write RAM and ROM Value of Parameter by UPID [Inputs used: UPIDIn, ValueIn]
 							Mode 5: Get minimal Value of Parameter by UPID [Inputs used: UPIDIn]
 							Mode 6: Get maximal Value of Parameter by UPID [Inputs used: UPIDIn]
 							Mode 7: Get default Value of Parameter by UPID [Inputs used: UPIDIn]
							*)
	UPIDIn			:UINT;	(*UPID to access*)
	ValueIn			:DINT;	(*UPID value to be written*)
	Streaming		:BOOL;	(*If enabled UPID is cyclically read / written. Only available for mode 1 & 3*)
END_VAR
VAR_IN_OUT
	Axis				:tstLM_Axis; (*Axis reference*)
END_VAR
VAR_OUTPUT
	Done			:BOOL;	(*Command has been executed*)
	Busy			:BOOL;	(*Command running / FB Busy*)
	ValueOut			:DINT;	(*UPID value from drive*)
	Error			:BOOL;	(*Error occured in FB*)
	ErrorID			:UINT;	(*Error ID:
							01h: Timeout (No Response from the drive)
							02h: ConfigChannel already busy
							03h: Invalid Mode selected
 							C0h: UPID Error 
 							C1h: Parameter Type Error
 							C2h: Range Error
 							C3h: Address Usage Error
 							C5h: Error: Command 21h
 							D0h: Odd Address
 							D1h: Size Error (Curve Service)
 							D4h: Curve already defined / Curve not present (Curve Service)
							>D4h: Contact LinMot Support
							*)
END_VAR
VAR
	uiState			:UINT;	(*internal -> *)
	uiStartState		:UINT;	(*internal -> *)
	fStartTrig			:LM_R_TRIG;	(*internal -> *)
	fTimer			:TON;	(*internal -> *)
	tiT1				:TIME:=T#5000ms; (*internal -> timeout*)
END_VAR
(*Version history:
Date         	 | Version    	| Created under     		| Author          		| Remark 
------------------------------------------------------------------------------------------------------------------------------- 
2011-jul-12   	 | 1.0.0      		| V2.11.0 (Build 1016)	| fj  				| initial release 
*)

(*Check on errors*)
IF ((SHR(Axis.DrvToPlc.CfgStatusWord,8) = 16#C0)
	OR (SHR(Axis.DrvToPlc.CfgStatusWord,8) = 16#C1)
	OR (SHR(Axis.DrvToPlc.CfgStatusWord,8) = 16#C2)
	OR (SHR(Axis.DrvToPlc.CfgStatusWord,8) = 16#C3)
	OR (SHR(Axis.DrvToPlc.CfgStatusWord,8) = 16#C5)
	OR (SHR(Axis.DrvToPlc.CfgStatusWord,8) = 16#D0)
	OR (SHR(Axis.DrvToPlc.CfgStatusWord,8) = 16#D1)
	OR (SHR(Axis.DrvToPlc.CfgStatusWord,8) = 16#D4)
	OR (SHR(Axis.DrvToPlc.CfgStatusWord,8) > 16#D4))
	AND uiState > 1
	AND Busy THEN
	ErrorID := SHR(Axis.DrvToPlc.CfgStatusWord, 8);
	uiState := 90;
END_IF

(*Mode selection and edge detection*)
fStartTrig(CLK:=Execute);
IF fStartTrig.Q AND NOT Busy THEN
	CASE Mode OF
		(*Read ROM Value of Parameter by UPID*)
		0: 	uiStartState := 2;
			uiState := 1;
		(*Read RAM Value of Parameter by UPID*)
		1: 	IF Streaming THEN
				uiStartState := 80; (*-> Streaming active*)
			ELSE
				uiStartState := 10; (*Single read*)
			END_IF
			uiState := 1;
		(*Write ROM Value of Parameter by UPID*)
		2: 	uiStartState := 20;
			uiState := 1;
		(*Write RAM Value of Parameter by UPID*)
		3: 	IF Streaming THEN
				uiStartState := 80; (*-> Streaming active*)
			ELSE
				uiStartState := 30; (*Single write*)
			END_IF
			uiState := 1;
		(*Write RAM and ROM Value of Parameter by UPID*)
		4: 	uiStartState := 40;
			uiState := 1;
		(*Get minimal Value of Parameter by UPID*)
		5: 	uiStartState := 50;
			uiState := 1;
		(*Get maximal Value of Parameter by UPID*)
		6: 	uiStartState := 60;
			uiState := 1;
		(*Get default Value of Parameter by UPID*)
		7: 	uiStartState := 70;
			uiState := 1;
		ELSE ;
	END_CASE

	IF Axis.ConfigChannelBusy THEN (*Check ConfigChannel busy*)
		ErrorID := 16#02; (*Error: ConfigChannel already busy*)
		uiState := 90; (*Error*)
	ELSIF Mode > 7 THEN
		ErrorID := 16#03; (*Error: Invalid Mode selected*)
		uiState := 90; (*Error*)
	ELSE
		Axis.ConfigChannelBusy := TRUE;
		Busy := TRUE;
	END_IF
END_IF

(*State machine*)
CASE uiState OF
	(*Idle state*)
	0: 	;

	(*Prepare Config Module*)
	1: 	Axis.PlcToDrv.CfgControlWord := 16#000F;
		Axis.PlcToDrv.CfgIndexOut := 16#0000;
		Axis.PlcToDrv.CfgValueOut := 16#00000000;
		fTimer(IN:=TRUE,PT:=tiT1);

		IF fTimer.Q THEN
			fTimer(IN:=FALSE);
			ErrorID := 16#01; (*fTimer error: No response from drive*)
			uiState := 90;
		END_IF

		IF Axis.DrvToPlc.CfgStatusWord = 16#000F THEN
			fTimer(IN:=FALSE);
			uiState := uiStartState;
		END_IF

(*=============================================================================
*  Mode 0: 
*  Read ROM Value of Parameter by UPID
===============================================================================*)    

	 (*Read ROM Value of Parameter by UPID*)
	2:	Axis.PlcToDrv.CfgControlWord := 16#1001;
		Axis.PlcToDrv.CfgIndexOut := UPIDIn;
		fTimer(IN:=TRUE,PT:=tiT1);

		IF fTimer.Q THEN
			fTimer(IN:=FALSE);
			ErrorID := 16#01; (*fTimer error: No response from drive*)
			uiState := 90;
		END_IF

		IF Axis.DrvToPlc.CfgStatusWord = 16#0001 THEN
			ValueOut := UDINT_TO_DINT(Axis.DrvToPlc.CfgValueIn);
			fTimer(IN:=FALSE);
			uiState := 100;
		END_IF

(*=============================================================================
*  Mode 1: 
*  Read RAM Value of Parameter by UPID
===============================================================================*)    

	 (*Read RAM Value of Parameter by UPID*)
	10:	Axis.PlcToDrv.CfgControlWord := 16#1101;
		Axis.PlcToDrv.CfgIndexOut := UPIDIn;
		fTimer(IN:=TRUE,PT:=tiT1);

		IF fTimer.Q THEN
			fTimer(IN:=FALSE);
			ErrorID := 16#01; (*fTimer error: No response from drive*)
			uiState := 90;
		END_IF

		IF Axis.DrvToPlc.CfgStatusWord = 16#0001THEN
			fTimer(IN:=FALSE);
			ValueOut := UDINT_TO_DINT(Axis.DrvToPlc.CfgValueIn);
			uiState := 100;
		END_IF

(*=============================================================================
*  Mode 2: 
*  Write ROM Value of Parameter by UPID
===============================================================================*)    

	 (*Write ROM Value of Parameter by UPID*)
	20:	Axis.PlcToDrv.CfgControlWord := 16#1201;
		Axis.PlcToDrv.CfgIndexOut := UPIDIn;
		Axis.PlcToDrv.CfgValueOut := DINT_TO_UDINT(ValueIn);
		fTimer(IN:=TRUE,PT:=tiT1);

		IF fTimer.Q THEN
			fTimer(IN:=FALSE);
			ErrorID := 16#01; (*fTimer error: No response from drive*)
			uiState := 90;
		END_IF

		IF Axis.DrvToPlc.CfgStatusWord = 16#0001 THEN
			fTimer(IN:=FALSE);
			ValueOut := UDINT_TO_DINT(Axis.DrvToPlc.CfgValueIn);
			uiState := 100;
		END_IF

(*=============================================================================
*  Mode 3: 
*  Write RAM Value of Parameter by UPID
===============================================================================*)    

	 (*Write RAM Value of Parameter by UPID*)
	30:	Axis.PlcToDrv.CfgControlWord := 16#1301;
		Axis.PlcToDrv.CfgIndexOut := UPIDIn;
		Axis.PlcToDrv.CfgValueOut := DINT_TO_UDINT(ValueIn);
		fTimer(IN:=TRUE,PT:=tiT1);

		IF fTimer.Q THEN
			fTimer(IN:=FALSE);
			ErrorID := 16#01; (*fTimer error: No response from drive*)
			uiState := 90;
		END_IF

		IF Axis.DrvToPlc.CfgStatusWord = 16#0001 THEN
			fTimer(IN:=FALSE);
			ValueOut := UDINT_TO_DINT(Axis.DrvToPlc.CfgValueIn);
			uiState := 100;
		END_IF

(*=============================================================================
*  Mode 4: 
*  Write RAM and ROM Value of Parameter by UPID
===============================================================================*)    

	 (*Write RAM and ROM Value of Parameter by UPID*)
	40:	Axis.PlcToDrv.CfgControlWord := 16#1401;
		Axis.PlcToDrv.CfgIndexOut :=  UPIDIn;
		Axis.PlcToDrv.CfgValueOut := DINT_TO_UDINT(ValueIn);
		fTimer(IN:=TRUE,PT:=tiT1);

		IF fTimer.Q THEN
			fTimer(IN:=FALSE);
			ErrorID := 16#01; (*fTimer error: No response from drive*)
			uiState := 90;
		END_IF

		IF Axis.DrvToPlc.CfgStatusWord = 16#0001 THEN
			fTimer(IN:=FALSE);
			ValueOut := UDINT_TO_DINT(Axis.DrvToPlc.CfgValueIn);
			uiState := 100;
		END_IF

(*=============================================================================
*  Mode 5: 
* Get minimal Value of Parameter by UPID
===============================================================================*)    

	(*Get minimal Value of Parameter by UPID*)
	50:	Axis.PlcToDrv.CfgControlWord := 16#1501;
		Axis.PlcToDrv.CfgIndexOut := UPIDIn;
		fTimer(IN:=TRUE,PT:=tiT1);

		IF fTimer.Q THEN
			fTimer(IN:=FALSE);
			ErrorID := 16#01; (*fTimer error: No response from drive*)
			uiState := 90;
		END_IF

		IF Axis.DrvToPlc.CfgStatusWord = 16#0001 THEN
			fTimer(IN:=FALSE);
			ValueOut := UDINT_TO_DINT(Axis.DrvToPlc.CfgValueIn);
			uiState := 100;
		END_IF

(*=============================================================================
*  Mode 6: 
* Get maximal Value of Parameter by UPID
===============================================================================*)    

	 (*Get maximal Value of Parameter by UPID*)
	60:	Axis.PlcToDrv.CfgControlWord := 16#1601;
		Axis.PlcToDrv.CfgIndexOut := UPIDIn;
		fTimer(IN:=TRUE,PT:=tiT1);

		IF fTimer.Q THEN
			fTimer(IN:=FALSE);
			ErrorID := 16#01; (*fTimer error: No response from drive*)
			uiState := 90;
		END_IF

		IF Axis.DrvToPlc.CfgStatusWord = 16#0001 THEN
			fTimer(IN:=FALSE);
			ValueOut := UDINT_TO_DINT(Axis.DrvToPlc.CfgValueIn);
			uiState := 100;
		END_IF

(*=============================================================================
*  Mode 7: 
* Get default Value of Parameter by UPID
===============================================================================*)    

	 (*Get default Value of Parameter by UPID*)
	70:	Axis.PlcToDrv.CfgControlWord := 16#1701;
		Axis.PlcToDrv.CfgIndexOut := UPIDIn;
		fTimer(IN:=TRUE,PT:=tiT1);

		IF fTimer.Q THEN
			fTimer(IN:=FALSE);
			ErrorID := 16#01; (*fTimer error: No response from drive*)
			uiState := 90;
		END_IF

		IF Axis.DrvToPlc.CfgStatusWord = 16#0001 THEN
			fTimer(IN:=FALSE);
			ValueOut := UDINT_TO_DINT(Axis.DrvToPlc.CfgValueIn);
			uiState := 100;
		END_IF

(*=============================================================================
*  Streaming: 
*  Read / Write a parameter cyclically from / to RAM
===============================================================================*)    

	 (*Send Command*)
	80:	IF Mode = 1 THEN (*Read RAM parameter*)
			IF Axis.PlcToDrv.CfgControlWord = 16#000F THEN
				Axis.PlcToDrv.CfgControlWord := 16#1100;
			END_IF
			Axis.PlcToDrv.CfgControlWord.0 := NOT Axis.PlcToDrv.CfgControlWord.0;
			Axis.PlcToDrv.CfgIndexOut := UPIDIn;
			ValueOut := UDINT_TO_DINT(Axis.DrvToPlc.CfgValueIn);
		ELSIF Mode = 3 THEN (*Write RAM parameter*)
			IF Axis.PlcToDrv.CfgControlWord = 16#000F THEN
				Axis.PlcToDrv.CfgControlWord := 16#1300;
			END_IF
			Axis.PlcToDrv.CfgControlWord.0 := NOT Axis.PlcToDrv.CfgControlWord.0;
			Axis.PlcToDrv.CfgIndexOut := UPIDIn;
			ValueOut := UDINT_TO_DINT(Axis.DrvToPlc.CfgValueIn);
		ELSIF NOT(Mode = 1 OR Mode = 3) THEN
			ErrorID := 16#03; (*Error: Invalid Mode selected*)
			uiState := 90; (*Error*)
		END_IF

		IF NOT Streaming OR NOT Execute THEN
			uiState := 100;
		END_IF

(*=============================================================================
*  Error State
===============================================================================*)    

	(*Error state I*)
	90:	IF Busy THEN
			Axis.ConfigChannelBusy := FALSE; (*Only reset ConfigChannelBusy if function block is Busy*)
			Axis.PlcToDrv.CfgControlWord := 16#0000; (*Reset Config Control*)
		END_IF

		Error := TRUE;
		Busy := FALSE;
		Done := FALSE;
		ValueOut := 0;
		fTimer(IN:=FALSE);

		uiState := 91;

	(*Error State II*)
	91:	IF NOT Execute THEN
			Error := FALSE;
			ErrorID := 0;
			uiState := 0;
		END_IF

(*=============================================================================
*  Command Done
===============================================================================*)    

	(*Command succesfully executed*)
	100:	Done := TRUE;
		Busy := FALSE;
		fTimer(IN:=FALSE);

		Axis.ConfigChannelBusy := FALSE;
		Axis.PlcToDrv.CfgControlWord := 16#0000; (*Reset Config Control*)

		uiState := 101;

	(*Wait Not Execute*)
	101:	IF NOT Execute THEN
			Done := FALSE;
			ValueOut := 0;
			uiState := 0;
		END_IF

END_CASE

END_FUNCTION_BLOCK

// POUs/LinMot Config Function Blocks/LMcf_CTAccess
FUNCTION_BLOCK LMcf_CTAccess
VAR_INPUT
	Execute			:BOOL;	(*Execute command*)
	Mode			:UINT;	(*Mode 0: Save to Flash [Inputs used: none]
 							Mode 1: Delete All Entries [Inputs used: none]
 							Mode 2: Delete Entry [Inputs used: CTID]
 							Mode 3: Write Entry [Inputs used: CTEntry]
 							Mode 4: Get Entry [Inputs used: CTEntry, CTID]
 							Mode 5: Get Presence List [Inputs used: PresenceList]
							*)
	CTID			:UINT; 	(*ID of the CT Entry to be read/written, only used in mode 2 and 4*)
END_VAR
VAR_IN_OUT
	Axis			:tstLM_Axis; (*Axis reference*)
	CTEntry			:tstLM_CfgCTEntry; (*LinMot Command Table Entry element -> see data types*)
	PresenceList	:ARRAY[0..7] OF UDINT; (*The presence list shows which lines of the command table are defined*)
END_VAR
VAR_OUTPUT
	Done			:BOOL;	(*Command has been executed*)
	Busy			:BOOL;	(*Command running / FB Busy*)
	Error			:BOOL;	(*Error occured in FB*)
	ErrorID			:UINT;	(*Error ID:
							01h: Timeout (No Response from the drive)
							02h: ConfigChannel already busy
							03h: Invalid Mode selected
 							C0h: UPID Error 
 							C1h: Parameter Type Error
 							C2h: Range Error
 							C3h: Address Usage Error
 							C5h: Error: Command 21h
 							D0h: Odd Address
 							D1h: Size Error (Curve Service)
 							D4h: Curve already defined / Curve not present (Curve Service)
							>D4h: Contact LinMot Support
							*)
END_VAR
VAR
	uiState			:UINT;	(*internal -> *)
	uiStartState	:UINT;	(*internal -> *)
	i				:UINT;	(*internal -> *)
	fStartTrig	:LM_R_TRIG	(*internal -> *);
	fTimer			:TON;	(*internal -> *)
	tiT1			:TIME:=T#5000MS; (*internal -> timout short*)
	tiT2			:TIME:=T#60000MS; (*internal -> timeout long*)
END_VAR
(*Version history:
Date         	 | Version    	| Created under     		| Author          		| Remark 
------------------------------------------------------------------------------------------------------------------------------- 
2011-jul-12   	 | 1.0.0      		| V2.11.0 (Build 1016)	| fj  				| initial release 
2012-aug-21   	 | 1.1.0      		| V2.11.0 (Build 1016)	| fj  				| in mode 4 (Get Entry) the last value was not read, fixed
*)

(*Check on errors*)
IF ((SHR(Axis.DrvToPlc.CfgStatusWord,8) = 16#C0)
	OR (SHR(Axis.DrvToPlc.CfgStatusWord,8) = 16#C1)
	OR (SHR(Axis.DrvToPlc.CfgStatusWord,8) = 16#C2)
	OR (SHR(Axis.DrvToPlc.CfgStatusWord,8) = 16#C3)
	OR (SHR(Axis.DrvToPlc.CfgStatusWord,8) = 16#C5)
	OR (SHR(Axis.DrvToPlc.CfgStatusWord,8) = 16#D0)
	OR (SHR(Axis.DrvToPlc.CfgStatusWord,8) = 16#D1)
	OR (SHR(Axis.DrvToPlc.CfgStatusWord,8) = 16#D4)
	OR (SHR(Axis.DrvToPlc.CfgStatusWord,8) > 16#D4))
	AND uiState > 1
	AND Busy THEN
	ErrorID := SHR(Axis.DrvToPlc.CfgStatusWord, 8);
	uiState := 90;
END_IF

(*Mode selection and edge detection*)
fStartTrig(CLK:=Execute);
IF fStartTrig.Q AND NOT Busy THEN
	CASE Mode OF
		(*Save to Flash*)
		0: 	uiStartState := 2;
			uiState := 1;
		(*Delete All Entries*)
		1: 	uiStartState := 10;
			uiState := 1;
		(*Delete Entry*)
		2: 	uiStartState := 20;
			uiState := 1;
		(*Write Entry*)
		3: 	uiStartState := 30;
			uiState := 1;
		(*Get Entry*)
		4: 	uiStartState := 40;
			uiState := 1;
		(*Get Presence List*)
		5: 	uiStartState := 50;
			uiState := 1;
		ELSE ;
	END_CASE
	IF Axis.ConfigChannelBusy THEN (*Check ConfigChannel busy*)
		ErrorID := 16#02; (*Error: ConfigChannel already busy*)
		uiState := 90; (*Error*)
	ELSIF Mode > 5 THEN
		ErrorID := 16#03; (*Error: Invalid Mode selected*)
		uiState := 90; (*Error*)
	ELSE
		Axis.ConfigChannelBusy := TRUE;
		Busy := TRUE;
	END_IF
END_IF

(*State machine*)
CASE uiState OF
	(*Idle state*)
	0: 	;

	(*Prepare Config Module*)
	1: 	Axis.PlcToDrv.CfgControlWord := 16#000F;
		Axis.PlcToDrv.CfgIndexOut := 16#0000;
		Axis.PlcToDrv.CfgValueOut := 16#00000000;
		fTimer(IN:=TRUE,PT:=tiT1);

		IF fTimer.Q THEN
			fTimer(IN:=FALSE);
			ErrorID := 16#01; (*fTimer error: No response from drive*)
			uiState := 90;
		END_IF

		IF Axis.DrvToPlc.CfgStatusWord = 16#000F THEN
			fTimer(IN:=FALSE);
			uiState := uiStartState; (*Jump to state selected by mode input*)
		END_IF

(*=============================================================================
*  Mode 0: 
*  Save to Flash
*  Note: 	MC software must  be stopped!! (not implemented here)
*		Use function block StopStartDefault
===============================================================================*)    

	 (*Save to Flash*)
	2:	Axis.PlcToDrv.CfgControlWord := 16#8001;
		fTimer(IN:=TRUE,PT:=tiT2);

		IF fTimer.Q THEN
			fTimer(IN:=FALSE);
			ErrorID := 16#01; (*fTimer error: No response from drive*)
			uiState := 90;
		END_IF

		IF Axis.DrvToPlc.CfgStatusWord = 16#0001 THEN
			fTimer(IN:=FALSE);
			uiState := 100;
		END_IF

(*=============================================================================
*  Mode 1: 
*  Delete All Entries (RAM)
===============================================================================*)    

	 (*Delete All Entries (RAM)*)
	10:	Axis.PlcToDrv.CfgControlWord := 16#8101;
		fTimer(IN:=TRUE,PT:=tiT2);

		IF fTimer.Q THEN
			fTimer(IN:=FALSE);
			ErrorID := 16#01; (*fTimer error: No response from drive*)
			uiState := 90;
		END_IF

		IF Axis.DrvToPlc.CfgStatusWord = 16#0001 THEN
			fTimer(IN:=FALSE);
			uiState := 100;
		END_IF

(*=============================================================================
*  Mode 2: 
*  Delete Entry
===============================================================================*)    

	 (*Delete Entry*)
	20:	Axis.PlcToDrv.CfgControlWord := 16#8201;
		Axis.PlcToDrv.CfgIndexOut := CTID;
		fTimer(IN:=TRUE,PT:=tiT1);

		IF fTimer.Q THEN
			fTimer(IN:=FALSE);
			ErrorID := 16#01; (*fTimer error: No response from drive*)
			uiState := 90;
		END_IF

		IF Axis.DrvToPlc.CfgStatusWord = 16#0001 THEN
			fTimer(IN:=FALSE);
			uiState := 100;
		END_IF

(*=============================================================================
*  Mode 3: 
*  Write Entry
===============================================================================*)    

	 (*Write Entry*)
	30:	Axis.PlcToDrv.CfgControlWord := 16#8301;
		Axis.PlcToDrv.CfgIndexOut := CTEntry.CTID; (*Entry ID*)
		Axis.PlcToDrv.CfgValueOut := CTEntry.BlockSize; (*Entry Block Size*)
		fTimer(IN:=TRUE,PT:=tiT1);

		IF fTimer.Q THEN
			fTimer(IN:=FALSE);
			ErrorID := 16#01; (*fTimer error: No response from drive*)
			uiState := 90;
		END_IF

		IF Axis.DrvToPlc.CfgStatusWord = 16#0001 THEN
			fTimer(IN:=FALSE);
			uiState := 31;
		END_IF

	 (*Write Entry Data*)
	31:	Axis.PlcToDrv.CfgControlWord := 16#8402;
		Axis.PlcToDrv.CfgIndexOut := CTEntry.CTID; (*Entry ID*)
		Axis.PlcToDrv.CfgValueOut := CTEntry.DataBlock[i];
		fTimer(IN:=TRUE,PT:=tiT1);

		IF fTimer.Q THEN
			fTimer(IN:=FALSE);
			ErrorID := 16#01; (*fTimer error: No response from drive*)
			uiState := 90;
		END_IF

		IF Axis.DrvToPlc.CfgStatusWord = 16#0002 THEN (*Block finished*)
			fTimer(IN:=FALSE);
			i := 0; (*Reset i*)
			uiState := 100;
		ELSIF Axis.DrvToPlc.CfgStatusWord = 16#0402 THEN (**)
			fTimer(IN:=FALSE);
			i := i+1;
			uiState := 32;
		END_IF

	(*Write Entry Data*)
	32:	Axis.PlcToDrv.CfgControlWord := 16#8403;
		Axis.PlcToDrv.CfgIndexOut := CTEntry.CTID; (*Entry ID*)
		Axis.PlcToDrv.CfgValueOut := CTEntry.DataBlock[i];
		fTimer(IN:=TRUE,PT:=tiT1);

		IF fTimer.Q THEN
			fTimer(IN:=FALSE);
			ErrorID := 16#01; (*fTimer error: No response from drive*)
			uiState := 90;
		END_IF

		IF Axis.DrvToPlc.CfgStatusWord = 16#0003 THEN (*Block finished*)
			fTimer(IN:=FALSE);
			i := 0; (*Reset i*)
			uiState := 100;
		ELSIF Axis.DrvToPlc.CfgStatusWord = 16#0403 THEN (**)
			fTimer(IN:=FALSE);
			i := i+1;
			uiState := 31;
		END_IF

(*=============================================================================
*  Mode 4: 
*  Get Entry
===============================================================================*)    

	 (*Get Entry*)
	40:	Axis.PlcToDrv.CfgControlWord := 16#8501;
		Axis.PlcToDrv.CfgIndexOut := CTID;
		fTimer(IN:=TRUE,PT:=tiT1);

		IF fTimer.Q THEN
			fTimer(IN:=FALSE);
			ErrorID := 16#01; (*fTimer error: No response from drive*)
			uiState := 90;
		END_IF

		IF Axis.DrvToPlc.CfgStatusWord = 16#0001 THEN
			fTimer(IN:=FALSE);
			CTEntry.CTID := Axis.DrvToPlc.CfgIndexIn;
			CTEntry.BlockSize := UDINT_TO_UINT(Axis.DrvToPlc.CfgValueIn);
			uiState := 41;
		END_IF

	 (*Get Entry Data*)
	41:	Axis.PlcToDrv.CfgControlWord := 16#8602;
		Axis.PlcToDrv.CfgIndexOut := CTID;
		fTimer(IN:=TRUE,PT:=tiT1);

		IF fTimer.Q THEN
			fTimer(IN:=FALSE);
			ErrorID := 16#01; (*fTimer error: No response from drive*)
			uiState := 90;
		END_IF

		IF Axis.DrvToPlc.CfgStatusWord = 16#0002 THEN (*Block finished*)
			fTimer(IN:=FALSE);
			CTEntry.DataBlock[i] := Axis.DrvToPlc.CfgValueIn; (*Read last Value*)
			i := 0; (*Reset i*)
			uiState := 100;
		ELSIF Axis.DrvToPlc.CfgStatusWord = 16#0402 THEN (*New data available*)
			fTimer(IN:=FALSE);
			CTEntry.DataBlock[i] := Axis.DrvToPlc.CfgValueIn; (*Read Value*)
			i := i+1;
			uiState := 42;
		END_IF

	(*Get Entry Data*)
	42:	Axis.PlcToDrv.CfgControlWord := 16#8603;
		Axis.PlcToDrv.CfgIndexOut := CTID;
		fTimer(IN:=TRUE,PT:=tiT1);

		IF fTimer.Q THEN
			fTimer(IN:=FALSE);
			ErrorID := 16#01; (*fTimer error: No response from drive*)
			uiState := 90;
		END_IF

		IF Axis.DrvToPlc.CfgStatusWord = 16#0003 THEN (*Block finished*)
			fTimer(IN:=FALSE);
			CTEntry.DataBlock[i] := Axis.DrvToPlc.CfgValueIn; (*Read last Value*)
			i := 0; (*Reset i*)
			uiState := 100;
		ELSIF Axis.DrvToPlc.CfgStatusWord = 16#0403 THEN (*New data vailable*)
			fTimer(IN:=FALSE);
			CTEntry.DataBlock[i] := Axis.DrvToPlc.CfgValueIn; (*Read Value*)
			i := i+1;
			uiState := 41;
		END_IF

(*=============================================================================
*  Mode 5: 
*  Get Presence List
===============================================================================*)    

	(*Get Presence List of Entries 0..31 from RAM*)
	50:	Axis.PlcToDrv.CfgControlWord := 16#8701;
		fTimer(IN:=TRUE,PT:=tiT1);

		IF fTimer.Q THEN
			fTimer(IN:=FALSE);
			ErrorID := 16#01; (*fTimer error: No response from drive*)
			uiState := 90;
		END_IF

		IF Axis.DrvToPlc.CfgStatusWord = 16#0001 THEN
			fTimer(IN:=FALSE);
			PresenceList[0] := Axis.DrvToPlc.CfgValueIn;
			uiState := 51;
		END_IF

	(*Get Presence List of Entries 32..63 from RAM*)
	51:	Axis.PlcToDrv.CfgControlWord := 16#8802;
		fTimer(IN:=TRUE,PT:=tiT1);

		IF fTimer.Q THEN
			fTimer(IN:=FALSE);
			ErrorID := 16#01; (*fTimer error: No response from drive*)
			uiState := 90;
		END_IF

		IF Axis.DrvToPlc.CfgStatusWord = 16#0002 THEN
			fTimer(IN:=FALSE);
			PresenceList[1] := Axis.DrvToPlc.CfgValueIn;
			uiState := 52;
		END_IF

	(*Get Presence List of Entries 64..95 from RAM*)
	52:	Axis.PlcToDrv.CfgControlWord := 16#8903;
		fTimer(IN:=TRUE,PT:=tiT1);

		IF fTimer.Q THEN
			fTimer(IN:=FALSE);
			ErrorID := 16#01; (*fTimer error: No response from drive*)
			uiState := 90;
		END_IF

		IF Axis.DrvToPlc.CfgStatusWord = 16#0003 THEN
			fTimer(IN:=FALSE);
			PresenceList[2] := Axis.DrvToPlc.CfgValueIn;
			uiState := 53;
		END_IF

	(*Get Presence List of Entries 96..127 from RAM*)
	53:	Axis.PlcToDrv.CfgControlWord := 16#8A04;
		fTimer(IN:=TRUE,PT:=tiT1);

		IF fTimer.Q THEN
			fTimer(IN:=FALSE);
			ErrorID := 16#01; (*fTimer error: No response from drive*)
			uiState := 90;
		END_IF

		IF Axis.DrvToPlc.CfgStatusWord = 16#0004 THEN
			fTimer(IN:=FALSE);
			PresenceList[3] := Axis.DrvToPlc.CfgValueIn;
			uiState := 54;
		END_IF

	(*Get Presence List of Entries 128..159 from RAM*)
	54:	Axis.PlcToDrv.CfgControlWord := 16#8B05;
		fTimer(IN:=TRUE,PT:=tiT1);

		IF fTimer.Q THEN
			fTimer(IN:=FALSE);
			ErrorID := 16#01; (*fTimer error: No response from drive*)
			uiState := 90;
		END_IF

		IF Axis.DrvToPlc.CfgStatusWord = 16#0005 THEN
			fTimer(IN:=FALSE);
			PresenceList[4] := Axis.DrvToPlc.CfgValueIn;
			uiState := 55;
		END_IF

	(*Get Presence List of Entries 160..191 from RAM*)
	55:	Axis.PlcToDrv.CfgControlWord := 16#8C06;
		fTimer(IN:=TRUE,PT:=tiT1);

		IF fTimer.Q THEN
			fTimer(IN:=FALSE);
			ErrorID := 16#01; (*fTimer error: No response from drive*)
			uiState := 90;
		END_IF

		IF Axis.DrvToPlc.CfgStatusWord = 16#0006 THEN
			fTimer(IN:=FALSE);
			PresenceList[5] := Axis.DrvToPlc.CfgValueIn;
			uiState := 56;
		END_IF

	(*Get Presence List of Entries 192..223 from RAM*)
	56:	Axis.PlcToDrv.CfgControlWord := 16#8D07;
		fTimer(IN:=TRUE,PT:=tiT1);

		IF fTimer.Q THEN
			fTimer(IN:=FALSE);
			ErrorID := 16#01; (*fTimer error: No response from drive*)
			uiState := 90;
		END_IF

		IF Axis.DrvToPlc.CfgStatusWord = 16#0007 THEN
			fTimer(IN:=FALSE);
			PresenceList[6] := Axis.DrvToPlc.CfgValueIn;
			uiState := 57;
		END_IF

	(*Get Presence List of Entries 223..255 from RAM*)
	57:	Axis.PlcToDrv.CfgControlWord := 16#8E08;
		fTimer(IN:=TRUE,PT:=tiT1);

		IF fTimer.Q THEN
			fTimer(IN:=FALSE);
			ErrorID := 16#01; (*fTimer error: No response from drive*)
			uiState := 90;
		END_IF

		IF Axis.DrvToPlc.CfgStatusWord = 16#0008 THEN
			fTimer(IN:=FALSE);
			PresenceList[7] := Axis.DrvToPlc.CfgValueIn;
			uiState := 100;
		END_IF

(*=============================================================================
*  Error State
===============================================================================*)    

	(*Error State I*)
	90:	IF Busy THEN
			Axis.ConfigChannelBusy := FALSE; (*Only reset ConfigChannelBusy if function block is Busy*)
			Axis.PlcToDrv.CfgControlWord := 16#0000; (*Reset Config Control*)
		END_IF

		Error := TRUE;
		Busy := FALSE;
		Done := FALSE;
		fTimer(IN:=FALSE);
		i := 0;

		uiState := 91;

	(*Error State II*)
	91:	IF NOT Execute THEN
			Error := FALSE;
			ErrorID := 0;
			uiState := 0;
		END_IF

(*=============================================================================
*  Command Done
===============================================================================*)    

	(*Command succesfully executed*)
	100:Done := TRUE;
		Busy := FALSE;
		fTimer(IN:=FALSE);
		i := 0;

		Axis.ConfigChannelBusy := FALSE;
		Axis.PlcToDrv.CfgControlWord := 16#0000; (*Reset Config Control*)

		uiState := 101;

	(*Wait Not Execute*)
	101:IF NOT Execute THEN
			Done := FALSE;
			uiState := 0;
		END_IF

END_CASE

END_FUNCTION_BLOCK

// POUs/LinMot Config Function Blocks/LMcf_CurveAccess
FUNCTION_BLOCK LMcf_CurveAccess
VAR_INPUT
	adrInfoBlock	:POINTER TO ARRAY[0..18] OF UDINT; (*Points to the start of the InfoBlock of a curve (motion profile)*)
	adrDataBlock	:POINTER TO UDINT; (*Points to the start of the DataBlock of a curve (motion profile)*)
	Execute			:BOOL;	(*Execute command*)
	Mode			:UINT;	(*Mode 0: Save all Curves from RAM to Flash [Inputs used: none]
 							Mode 1: Delete all curves (RAM) [Inputs used: none]
 							Mode 2: Add Curve (RAM) [Inputs used: CurveElement]
 							Mode 3: Modify Curve (RAM) [Inputs used: CurveElement]
 							Mode 4: Get Curve (RAM) [Inputs used: iCurveID, CurveElement]
							*)
	CurveID			:UINT; 	(*ID of the curve to be read*)
END_VAR
VAR_IN_OUT
	Axis			:tstLM_Axis; (*Axis reference*)
END_VAR
VAR_OUTPUT
	Done			:BOOL;	(*Command has been executed*)
	Busy			:BOOL;	(*Command running / FB Busy*)
	Error			:BOOL;	(*Error occured in FB*)
	ErrorID			:UINT;	(*Error ID:
							01h: Timeout (No Response from the drive)
							02h: ConfigChannel already busy
							03h: Invalid Mode selected
							04h: Address of adrDataBlock or adrInfoBlock is invalid (0), check inputs (CurveAccess)
 							C0h: UPID Error 
 							C1h: Parameter Type Error
 							C2h: Range Error
 							C3h: Address Usage Error
 							C5h: Error: Command 21h
 							D0h: Odd Address
 							D1h: Size Error (Curve Service)
 							D4h: Curve already defined / Curve not present (Curve Service)
							>D4h: Contact LinMot Support
							*)
END_VAR
VAR
	uiState			:UINT;	(*internal -> *)
	uiStartState	:UINT;	(*internal -> *)
	i				:UINT;	(*internal -> *)
	pDataBlock		:POINTER TO UDINT; (*internal -> *)
	fStartTrig		:LM_R_TRIG;	(*internal -> *)
	fTimer			:TON;	(*internal -> *)
	tiT1			:TIME:=T#5000MS;	(*internal -> timout short*)
	tiT2			:TIME:=T#60000MS; (*internal -> timeout long*)
END_VAR
(*Version history:
Date         	 | Version    	| Created under     		| Author          		| Remark 
------------------------------------------------------------------------------------------------------------------------------- 
2011-jul-12   	 | 1.0.0      		| V2.11.0 (Build 1016)	| fj  				| initial release 
*)

(*Check on errors*)
IF ((SHR(Axis.DrvToPlc.CfgStatusWord,8) = 16#C0)
	OR (SHR(Axis.DrvToPlc.CfgStatusWord,8) = 16#C1)
	OR (SHR(Axis.DrvToPlc.CfgStatusWord,8) = 16#C2)
	OR (SHR(Axis.DrvToPlc.CfgStatusWord,8) = 16#C3)
	OR (SHR(Axis.DrvToPlc.CfgStatusWord,8) = 16#C5)
	OR (SHR(Axis.DrvToPlc.CfgStatusWord,8) = 16#D0)
	OR (SHR(Axis.DrvToPlc.CfgStatusWord,8) = 16#D1)
	OR (SHR(Axis.DrvToPlc.CfgStatusWord,8) = 16#D4)
	OR (SHR(Axis.DrvToPlc.CfgStatusWord,8) > 16#D4))
	AND uiState > 1
	AND Busy THEN
	ErrorID := SHR(Axis.DrvToPlc.CfgStatusWord, 8);
	uiState := 90;
END_IF

(*Mode selection and edge detection*)
fStartTrig(CLK:=Execute);
IF fStartTrig.Q AND NOT Busy THEN
	CASE Mode OF
		(*Save all Curves from RAM to Flash*)
		0: 	uiStartState := 2;
			uiState := 1;
		(*Delete all Curves (RAM)*)
		1: 	uiStartState := 10;
			uiState := 1;
		(*Add Curve (RAM)*)
		2: 	uiStartState := 20;
			uiState := 1;
		(*Modify Curve (RAM)*)
		3: 	uiStartState := 30;
			uiState := 1;
		(*Get Curve (RAM)*)
		4: 	uiStartState := 40;
			uiState := 1;
		ELSE ;
	END_CASE
	IF Axis.ConfigChannelBusy THEN (*Check ConfigChannel busy*)
		ErrorID := 16#02; (*Error: ConfigChannel already busy*)
		uiState := 90; (*Error*)
	ELSIF Mode > 4 THEN
		ErrorID := 16#03; (*Error: Invalid Mode selected*)
		uiState := 90; (*Error*)
	ELSIF Mode > 1 AND ((adrDataBlock = 0) OR (adrInfoBlock = 0)) THEN
		ErrorID := 16#04; (*Error: Address of adrInfoBlock or adrDataBlock is invalid (0), check inputs (CurveAccess)*)
		uiState := 90; (*Error*)
	ELSE
		Axis.ConfigChannelBusy := TRUE;
		Busy := TRUE;
	END_IF
END_IF

(*State machine*)
CASE uiState OF
	(*Idle state*)
	0: 	;

	(*Prepare Config Module*)
	1: 	Axis.PlcToDrv.CfgControlWord := 16#000F;
		Axis.PlcToDrv.CfgIndexOut := 16#0000;
		Axis.PlcToDrv.CfgValueOut := 16#00000000;
		fTimer(IN:=TRUE,PT:=tiT1);
		i := 0;
		pDataBlock := adrDataBlock;

		IF fTimer.Q THEN
			fTimer(IN:=FALSE);
			ErrorID := 16#01; (*fTimer error: No response from drive*)
			uiState := 90;
		END_IF

		IF Axis.DrvToPlc.CfgStatusWord = 16#000F THEN
			fTimer(IN:=FALSE);
			uiState := uiStartState;
		END_IF

(*=============================================================================
*  Mode 0: 
*  Curve Service: Save all curves from RAM to Flash
*  Note: 	MC software must  be stopped!! (not implemented here)
*		Use function block StopStartDefault
===============================================================================*)    

	(*Save all curves from RAM to Flash.*)
	2:	Axis.PlcToDrv.CfgControlWord := 16#4001;

		fTimer(IN:=TRUE,PT:=tiT2);

		IF fTimer.Q THEN
			fTimer(IN:=FALSE);
			ErrorID := 16#01; (*fTimer error: No response from drive*)
			uiState := 90;
		END_IF

		IF Axis.DrvToPlc.CfgStatusWord = 16#0001 THEN
			fTimer(IN:=FALSE);
			uiState := 100;
		END_IF

(*=============================================================================
*  Mode 1: 
*  Curve Service: Delete all Curves (RAM)
*  Note: fTimer time may have to be modified. Actually 20'000ms
===============================================================================*)    

	(*Delete all curves*)
	10:	Axis.PlcToDrv.CfgControlWord := 16#4101;

		fTimer(IN:=TRUE,PT:=tiT2);

		IF fTimer.Q THEN
			fTimer(IN:=FALSE);
			ErrorID := 16#01; (*fTimer error: No response from drive*)
			uiState := 90;
		END_IF

		IF Axis.DrvToPlc.CfgStatusWord = 16#0001 THEN
			fTimer(IN:=FALSE);
			uiState := 100;
		END_IF

(*=============================================================================
*  Mode 2: 
*  Curve Service: Add Curve (RAM)
===============================================================================*)    

	(*Start adding curve*)
	20:	Axis.PlcToDrv.CfgControlWord := 16#5001;
		Axis.PlcToDrv.CfgIndexOut := UDINT_TO_UINT(SHR(adrInfoBlock^[7],16));  (*Curve ID to modify*)
		Axis.PlcToDrv.CfgValueOut := SHL(adrInfoBlock^[1]*4 ,16) + SHR(SHL(adrInfoBlock^[0], 16),16); (*Info and data block size*)
		fTimer(IN:=TRUE,PT:=tiT1);

		IF fTimer.Q THEN
			fTimer(IN:=FALSE);
			ErrorID := 16#01; (*fTimer error: No response from drive*)
			uiState := 90;
		END_IF

		IF Axis.DrvToPlc.CfgStatusWord = 16#0001 THEN
			fTimer(IN:=FALSE);
			uiState := 21;
		END_IF

	(*Add curve info block*)
	21:	Axis.PlcToDrv.CfgControlWord := 16#5102;
		Axis.PlcToDrv.CfgValueOut := adrInfoBlock^[i];
		fTimer(IN:=TRUE,PT:=tiT1);

		IF fTimer.Q THEN
			fTimer(IN:=FALSE);
			ErrorID := 16#01; (*fTimer error: No response from drive*)
			uiState := 90;
		END_IF

		IF Axis.DrvToPlc.CfgStatusWord = 16#0002 THEN (*Block finished (70 Bytes)*)
			fTimer(IN:=FALSE);
			i := 0; (*Reset i*)
			uiState := 23;
		ELSIF Axis.DrvToPlc.CfgStatusWord = 16#0402 THEN (**)
			fTimer(IN:=FALSE);
			i := i+1;
			uiState := 22;
		END_IF

	(*Add curve info block*)
	22:	Axis.PlcToDrv.CfgControlWord := 16#5103;
		Axis.PlcToDrv.CfgValueOut := adrInfoBlock^[i];
		fTimer(IN:=TRUE,PT:=tiT1);

		IF fTimer.Q THEN
			fTimer(IN:=FALSE);
			ErrorID := 16#01; (*fTimer error: No response from drive*)
			uiState := 90;
		END_IF

		IF Axis.DrvToPlc.CfgStatusWord = 16#0003 THEN (*Block finished (70 Bytes)*)
			fTimer(IN:=FALSE);
			i := 0; (*Reset i*)
			uiState := 23;
		ELSIF Axis.DrvToPlc.CfgStatusWord = 16#0403 THEN (**)
			fTimer(IN:=FALSE);
			i := i+1;
			uiState := 21;
		END_IF

	(*Add curve data*)
	23:	Axis.PlcToDrv.CfgControlWord := 16#5204;
		Axis.PlcToDrv.CfgValueOut := pDataBlock^;
		fTimer(IN:=TRUE,PT:=tiT1);

		IF fTimer.Q THEN
			fTimer(IN:=FALSE);
			ErrorID := 16#01; (*fTimer error: No response from drive*)
			uiState := 90;
		END_IF

		IF Axis.DrvToPlc.CfgStatusWord = 16#0004 THEN (*Block finished*)
			fTimer(IN:=FALSE);
			uiState := 100;
		ELSIF Axis.DrvToPlc.CfgStatusWord = 16#0404 THEN (**)
			fTimer(IN:=FALSE);
			pDataBlock := pDataBlock + (SIZEOF(adrDataBlock^));
			i := i+1;
			uiState := 24;
		END_IF

	(*Add curve data*)
	24:	Axis.PlcToDrv.CfgControlWord := 16#5205;
		Axis.PlcToDrv.CfgValueOut := pDataBlock^;
		fTimer(IN:=TRUE,PT:=tiT1);

		IF fTimer.Q THEN
			fTimer(IN:=FALSE);
			ErrorID := 16#01; (*fTimer error: No response from drive*)
			uiState := 90;
		END_IF

		IF Axis.DrvToPlc.CfgStatusWord = 16#0005 THEN (*Block finished*)
			fTimer(IN:=FALSE);
			uiState := 100;
		ELSIF Axis.DrvToPlc.CfgStatusWord = 16#0405 THEN (**)
			fTimer(IN:=FALSE);
			pDataBlock := pDataBlock + (SIZEOF(adrDataBlock^));
			i := i+1;
			uiState := 23;
		END_IF

(*=============================================================================
*  Mode 3: 
*  Curve Service: Modify Curve (RAM)
===============================================================================*)    

	(*Start modifying curve*)
	30:	Axis.PlcToDrv.CfgControlWord := 16#5301;
		Axis.PlcToDrv.CfgIndexOut := UDINT_TO_UINT(SHR(adrInfoBlock^[7],16)); (*Curve ID to modify*)
		Axis.PlcToDrv.CfgValueOut := SHL(adrInfoBlock^[1]*4 ,16) + SHR(SHL(adrInfoBlock^[0], 16),16); (*Info and data block size*)
		fTimer(IN:=TRUE,PT:=tiT1);

		IF fTimer.Q THEN
			fTimer(IN:=FALSE);
			ErrorID := 16#01; (*fTimer error: No response from drive*)
			uiState := 90;
		END_IF

		IF Axis.DrvToPlc.CfgStatusWord = 16#0001 THEN
			fTimer(IN:=FALSE);
			uiState := 31;
		END_IF

	(*Modify curve info block*)
	31:	Axis.PlcToDrv.CfgControlWord := 16#5402;
		Axis.PlcToDrv.CfgValueOut := adrInfoBlock^[i];
		fTimer(IN:=TRUE,PT:=tiT1);

		IF fTimer.Q THEN
			fTimer(IN:=FALSE);
			ErrorID := 16#01; (*fTimer error: No response from drive*)
			uiState := 90;
		END_IF

		IF Axis.DrvToPlc.CfgStatusWord = 16#0002 THEN (*Block finished*)
			fTimer(IN:=FALSE);
			i := 0; (*Reset i*)
			uiState := 33;
		ELSIF Axis.DrvToPlc.CfgStatusWord = 16#0402 THEN (**)
			fTimer(IN:=FALSE);
			i := i+1;
			uiState := 32;
		END_IF

	(*Modify curve info block*)
	32:	Axis.PlcToDrv.CfgControlWord := 16#5403;
		Axis.PlcToDrv.CfgValueOut := adrInfoBlock^[i];
		fTimer(IN:=TRUE,PT:=tiT1);

		IF fTimer.Q THEN
			fTimer(IN:=FALSE);
			ErrorID := 16#01; (*fTimer error: No response from drive*)
			uiState := 90;
		END_IF

		IF Axis.DrvToPlc.CfgStatusWord = 16#0003 THEN (*Block finished (70 Bytes)*)
			fTimer(IN:=FALSE);
			i := 0; (*Reset i*)
			uiState := 33;
		ELSIF Axis.DrvToPlc.CfgStatusWord = 16#0403 THEN (**)
			fTimer(IN:=FALSE);
			i := i+1;
			uiState := 31;
		END_IF

	(*Modify curve data block*)
	33:	Axis.PlcToDrv.CfgControlWord := 16#5504;
		Axis.PlcToDrv.CfgValueOut := pDataBlock^;
		fTimer(IN:=TRUE,PT:=tiT1);

		IF fTimer.Q THEN
			fTimer(IN:=FALSE);
			ErrorID := 16#01; (*fTimer error: No response from drive*)
			uiState := 90;
		END_IF

		IF Axis.DrvToPlc.CfgStatusWord = 16#0004 THEN (*Block finished*)
			fTimer(IN:=FALSE);
			uiState := 100;
		ELSIF Axis.DrvToPlc.CfgStatusWord = 16#0404 THEN (**)
			fTimer(IN:=FALSE);
			pDataBlock := pDataBlock + (SIZEOF(adrDataBlock^));
			i := i+1;
			uiState := 34;
		END_IF

	(*Modify curve data block*)
	34:	Axis.PlcToDrv.CfgControlWord := 16#5505;
		Axis.PlcToDrv.CfgValueOut := pDataBlock^;
		fTimer(IN:=TRUE,PT:=tiT1);

		IF fTimer.Q THEN
			fTimer(IN:=FALSE);
			ErrorID := 16#01; (*fTimer error: No response from drive*)
			uiState := 90;
		END_IF

		IF Axis.DrvToPlc.CfgStatusWord = 16#0005 THEN (*Block finished*)
			fTimer(IN:=FALSE);
			uiState := 100;
		ELSIF Axis.DrvToPlc.CfgStatusWord = 16#0405 THEN (**)
			fTimer(IN:=FALSE);
			pDataBlock := pDataBlock + (SIZEOF(adrDataBlock^));
			i := i+1;
			uiState := 33;
		END_IF

(*=============================================================================
*  Mode 4: 
*  Curve Service: Get Curve (RAM)
*  Note: The input iCurveID is only used in this mode
===============================================================================*)    

	(*Start getting curve*)
	40:	Axis.PlcToDrv.CfgControlWord := 16#6001;
		Axis.PlcToDrv.CfgIndexOut := CurveID;
		fTimer(IN:=TRUE,PT:=tiT1);

		IF fTimer.Q THEN
			fTimer(IN:=FALSE);
			ErrorID := 16#01; (*fTimer error: No response from drive*)
			uiState := 90;
		END_IF

		IF Axis.DrvToPlc.CfgStatusWord = 16#0001 THEN
			fTimer(IN:=FALSE);
			uiState := 41;
		END_IF

	(*Get curve info block*)
	41:	Axis.PlcToDrv.CfgControlWord := 16#6102;
		fTimer(IN:=TRUE,PT:=tiT1);

		IF fTimer.Q THEN
			fTimer(IN:=FALSE);
			ErrorID := 16#01; (*fTimer error: No response from drive*)
			uiState := 90;
		END_IF

		IF Axis.DrvToPlc.CfgStatusWord = 16#0002 THEN (*Block finished*)
			fTimer(IN:=FALSE);
			adrInfoBlock^[i] := Axis.DrvToPlc.CfgValueIn; (*Read last double word*)
			i := 0; (*Reset i*)
			uiState := 43;
		ELSIF Axis.DrvToPlc.CfgStatusWord = 16#0402 THEN (*Block not finished but new data available*)
			fTimer(IN:=FALSE);
			adrInfoBlock^[i] := Axis.DrvToPlc.CfgValueIn;
			i := i+1;
			uiState := 42;
		END_IF

	(*Get curve info block*)
	42:	Axis.PlcToDrv.CfgControlWord := 16#6103;
		fTimer(IN:=TRUE,PT:=tiT1);

		IF fTimer.Q THEN
			fTimer(IN:=FALSE);
			ErrorID := 16#01; (*fTimer error: No response from drive*)
			uiState := 90;
		END_IF

		IF Axis.DrvToPlc.CfgStatusWord = 16#0003 THEN (*Block finished*)
			fTimer(IN:=FALSE);
			adrInfoBlock^[i] := Axis.DrvToPlc.CfgValueIn; (*Read last double word*)
			i := 0; (*Reset i*)
			uiState := 43;
		ELSIF Axis.DrvToPlc.CfgStatusWord = 16#0403 THEN (*Block not finished but new data available*)
			fTimer(IN:=FALSE);
			adrInfoBlock^[i] := Axis.DrvToPlc.CfgValueIn;
			i := i+1;
			uiState := 41;
		END_IF

	(*Get curve data block*)
	43:	Axis.PlcToDrv.CfgControlWord := 16#6204;
		fTimer(IN:=TRUE,PT:=tiT1);

		IF fTimer.Q THEN
			fTimer(IN:=FALSE);
			ErrorID := 16#01; (*fTimer error: No response from drive*)
			uiState := 90;
		END_IF

		IF Axis.DrvToPlc.CfgStatusWord = 16#0004 THEN (*Block finished*)
			fTimer(IN:=FALSE);
			pDataBlock^ := Axis.DrvToPlc.CfgValueIn; (*Read last set point*)
			uiState := 100;
		ELSIF Axis.DrvToPlc.CfgStatusWord = 16#0404 THEN (*Block not finished but new data available*)
			fTimer(IN:=FALSE);
			pDataBlock^ := Axis.DrvToPlc.CfgValueIn;
			pDataBlock := pDataBlock + (SIZEOF(adrDataBlock^));
			i := i+1;
			uiState := 44;
		END_IF

	(*Get curve data block*)
	44:	Axis.PlcToDrv.CfgControlWord := 16#6205;
		fTimer(IN:=TRUE,PT:=tiT1);

		IF fTimer.Q THEN
			fTimer(IN:=FALSE);
			ErrorID := 16#01; (*fTimer error: No response from drive*)
			uiState := 90;
		END_IF

		IF Axis.DrvToPlc.CfgStatusWord = 16#0005 THEN (*Block finished*)
			fTimer(IN:=FALSE);
			pDatablock^ := Axis.DrvToPlc.CfgValueIn; (*Read last set point*)
			uiState := 100;
		ELSIF Axis.DrvToPlc.CfgStatusWord = 16#0405 THEN (*Block not finished but new data available*)
			fTimer(IN:=FALSE);
			pDataBlock^ := Axis.DrvToPlc.CfgValueIn;
			pDataBlock := pDataBlock + (SIZEOF(adrDataBlock^));
			i := i+1;
			uiState := 43;
		END_IF

(*=============================================================================
*  Error State
===============================================================================*)    

	(*Error State I*)
	90:	IF Busy THEN
			Axis.ConfigChannelBusy := FALSE; (*Only reset ConfigChannelBusy if function block is Busy*)
			Axis.PlcToDrv.CfgControlWord := 16#0000; (*Reset Config Control*)
		END_IF

		Error := TRUE;
		Busy := FALSE;
		Done := FALSE;
		fTimer(IN:=FALSE);
		i := 0;

		uiState := 91;

	(*Error State II*)
	91:	IF NOT Execute THEN
			Error := FALSE;
			ErrorID := 0;
			uiState := 0;
		END_IF

(*=============================================================================
*  Command Done
===============================================================================*)    

	(*Command succesfully executed*)
	100:	Done := TRUE;
		Busy := FALSE;
		fTimer(IN:=FALSE);
		i := 0;

		Axis.ConfigChannelBusy := FALSE;
		Axis.PlcToDrv.CfgControlWord := 16#0000; (*Reset Config Control*)

		uiState := 101;

	(*Wait Not Execute*)
	101:	IF NOT Execute THEN
			Done := FALSE;
			uiState := 0;
		END_IF

END_CASE

END_FUNCTION_BLOCK

// POUs/LinMot Config Function Blocks/LMcf_GetErrorTxt
FUNCTION_BLOCK LMcf_GetErrorTxt
VAR_INPUT
	Execute			:BOOL;	(*Execute command*)
	ErrorCode		:UINT;	(*Error ID from which the String should be read out*)
END_VAR
VAR_IN_OUT
	Axis			:tstLM_Axis; (*Axis reference*)
END_VAR
VAR_OUTPUT
	Done			:BOOL;	(*Command has been executed*)
	Busy			:BOOL;	(*Command running / FB Busy*)
	ErrorText		:STRING;(*Error Text of the corresponding ErrorCode*)
	Error			:BOOL;	(*Error occured in FB*)
	ErrorID			:UINT;	(*Error ID:
							01h: Timeout (No Response from the drive)
							02h: ConfigChannel already busy
 							C0h: UPID Error 
 							C1h: Parameter Type Error
 							C2h: Range Error
 							C3h: Address Usage Error
 							C5h: Error: Command 21h
 							D0h: Odd Address
 							D1h: Size Error (Curve Service)
 							D4h: Curve already defined / Curve not present (Curve Service)
							>D4h: Contact LinMot Support
							*)
END_VAR
VAR
	uiState			:UINT;	(*internal -> *)
	i				:UINT;	(*internal -> *)
	fStartTrig		:LM_R_TRIG;	(*internal -> *)
	fTimer			:TON;	(*internal -> *)
	tiT1			:TIME:=T#5000MS; (*internal -> timeout*)
	TextStringletsBA:ARRAY[0..31] OF USINT; (*internal -> *)
	TextStringletsS	:ARRAY[0..31] OF STRING; (*internal -> *)
END_VAR
(*Version history:
Date         	 | Version    	| Created under     		| Author          		| Remark 
------------------------------------------------------------------------------------------------------------------------------- 
2011-jul-12   	 | 1.0.0      		| V2.11.0 (Build 1016)	| fj  				| initial release 
*)

(*Check on errors*)
IF ((SHR(Axis.DrvToPlc.CfgStatusWord,8) = 16#C0)
	OR (SHR(Axis.DrvToPlc.CfgStatusWord,8) = 16#C1)
	OR (SHR(Axis.DrvToPlc.CfgStatusWord,8) = 16#C2)
	OR (SHR(Axis.DrvToPlc.CfgStatusWord,8) = 16#C3)
	OR (SHR(Axis.DrvToPlc.CfgStatusWord,8) = 16#C5)
	OR (SHR(Axis.DrvToPlc.CfgStatusWord,8) = 16#D0)
	OR (SHR(Axis.DrvToPlc.CfgStatusWord,8) = 16#D1)
	OR (SHR(Axis.DrvToPlc.CfgStatusWord,8) = 16#D4)
	OR (SHR(Axis.DrvToPlc.CfgStatusWord,8) > 16#D4))
	AND uiState > 1
	AND Busy THEN
	ErrorID := SHR(Axis.DrvToPlc.CfgStatusWord, 8);
	uiState := 90;
END_IF

(*Check start trigger*)
fStartTrig(CLK:=Execute);
IF fStartTrig.Q AND NOT Busy THEN
	IF Axis.ConfigChannelBusy THEN (*Check ConfigChannel busy*)
		ErrorID := 16#02; (*Error: ConfigChannel already busy*)
		uiState := 90; (*Error*)
	ELSE
		Axis.ConfigChannelBusy := TRUE;
		Busy := TRUE;
		uiState := 1;
	END_IF
END_IF

(*State machine*)
CASE uiState OF
	(*Idle state*)
	0: 	;

(*=============================================================================
*  Get ErrorCode Text
===============================================================================*)

	(*Prepare Config Module*)
	1: 	Axis.PlcToDrv.CfgControlWord := 16#000F;
		Axis.PlcToDrv.CfgIndexOut := 16#0000;
		Axis.PlcToDrv.CfgValueOut := 16#00000000;
		fTimer(IN:=TRUE,PT:=tiT1);

		IF fTimer.Q THEN
			fTimer(IN:=FALSE);
			ErrorID := 16#01; (*fTimer error: No response from drive*)
			uiState := 90;
		END_IF

		IF Axis.DrvToPlc.CfgStatusWord = 16#000F THEN
			fTimer(IN:=FALSE);
			uiState := 2;
		END_IF

	(*Get Stringlet 0*)
	2:	Axis.PlcToDrv.CfgControlWord := 16#7401;
		Axis.PlcToDrv.CfgIndexOut := ErrorCode;
		Axis.PlcToDrv.CfgValueOut := 0; (*Stringlet 0*)
		fTimer(IN:=TRUE,PT:=tiT1);

		IF fTimer.Q THEN
			fTimer(IN:=FALSE);
			ErrorID := 16#01; (*fTimer error: No response from drive*)
			uiState := 90;
		END_IF

		IF Axis.DrvToPlc.CfgStatusWord = 16#0001 THEN
			fTimer(IN:=FALSE);
			TextStringletsBA[0]:= UDINT_TO_USINT(Axis.DrvToPlc.CfgValueIn);
			TextStringletsBA[1]:= UDINT_TO_USINT(SHR(Axis.DrvToPlc.CfgValueIn,8));
			TextStringletsBA[2]:= UDINT_TO_USINT(SHR(Axis.DrvToPlc.CfgValueIn,16));
			TextStringletsBA[3]:= UDINT_TO_USINT(SHR(Axis.DrvToPlc.CfgValueIn,24));
			uiState := 3;
		END_IF

	(*Get Stringlet 1*)
	3:	Axis.PlcToDrv.CfgControlWord := 16#7402;
		Axis.PlcToDrv.CfgIndexOut := ErrorCode;
		Axis.PlcToDrv.CfgValueOut := 1; (*Stringlet 1*)
		fTimer(IN:=TRUE,PT:=tiT1);

		IF fTimer.Q THEN
			fTimer(IN:=FALSE);
			ErrorID := 16#01; (*fTimer error: No response from drive*)
			uiState := 90;
		END_IF

		IF Axis.DrvToPlc.CfgStatusWord = 16#0002 THEN
			fTimer(IN:=FALSE);
			TextStringletsBA[4]:= UDINT_TO_USINT(Axis.DrvToPlc.CfgValueIn);
			TextStringletsBA[5]:= UDINT_TO_USINT(SHR(Axis.DrvToPlc.CfgValueIn,8));
			TextStringletsBA[6]:= UDINT_TO_USINT(SHR(Axis.DrvToPlc.CfgValueIn,16));
			TextStringletsBA[7]:= UDINT_TO_USINT(SHR(Axis.DrvToPlc.CfgValueIn,24));
			uiState := 4;
		END_IF

	(*Get Stringlet 2*)
	4:	Axis.PlcToDrv.CfgControlWord := 16#7403;
		Axis.PlcToDrv.CfgIndexOut := ErrorCode;
		Axis.PlcToDrv.CfgValueOut := 2; (*Stringlet 2*)
		fTimer(IN:=TRUE,PT:=tiT1);

		IF fTimer.Q THEN
			fTimer(IN:=FALSE);
			ErrorID := 16#01; (*fTimer error: No response from drive*)
			uiState := 90;
		END_IF

		IF Axis.DrvToPlc.CfgStatusWord = 16#0003 THEN
			fTimer(IN:=FALSE);
			TextStringletsBA[8]:= UDINT_TO_USINT(Axis.DrvToPlc.CfgValueIn);
			TextStringletsBA[9]:= UDINT_TO_USINT(SHR(Axis.DrvToPlc.CfgValueIn,8));
			TextStringletsBA[10]:= UDINT_TO_USINT(SHR(Axis.DrvToPlc.CfgValueIn,16));
			TextStringletsBA[11]:= UDINT_TO_USINT(SHR(Axis.DrvToPlc.CfgValueIn,24));
			uiState := 5;
		END_IF

	(*Get Stringlet 3*)
	5:	Axis.PlcToDrv.CfgControlWord := 16#7404;
		Axis.PlcToDrv.CfgIndexOut := ErrorCode;
		Axis.PlcToDrv.CfgValueOut := 3; (*Stringlet 3*)
		fTimer(IN:=TRUE,PT:=tiT1);

		IF fTimer.Q THEN
			fTimer(IN:=FALSE);
			ErrorID := 16#01; (*fTimer error: No response from drive*)
			uiState := 90;
		END_IF

		IF Axis.DrvToPlc.CfgStatusWord = 16#0004 THEN
			fTimer(IN:=FALSE);
			TextStringletsBA[12]:= UDINT_TO_USINT(Axis.DrvToPlc.CfgValueIn);
			TextStringletsBA[13]:= UDINT_TO_USINT(SHR(Axis.DrvToPlc.CfgValueIn,8));
			TextStringletsBA[14]:= UDINT_TO_USINT(SHR(Axis.DrvToPlc.CfgValueIn,16));
			TextStringletsBA[15]:= UDINT_TO_USINT(SHR(Axis.DrvToPlc.CfgValueIn,24));
			uiState := 6;
		END_IF

	(*Get Stringlet 4*)
	6:	Axis.PlcToDrv.CfgControlWord := 16#7405;
		Axis.PlcToDrv.CfgIndexOut := ErrorCode;
		Axis.PlcToDrv.CfgValueOut := 4; (*Stringlet 4*)
		fTimer(IN:=TRUE,PT:=tiT1);

		IF fTimer.Q THEN
			fTimer(IN:=FALSE);
			ErrorID := 16#01; (*fTimer error: No response from drive*)
			uiState := 90;
		END_IF

		IF Axis.DrvToPlc.CfgStatusWord = 16#0005 THEN
			fTimer(IN:=FALSE);
			TextStringletsBA[16]:= UDINT_TO_USINT(Axis.DrvToPlc.CfgValueIn);
			TextStringletsBA[17]:= UDINT_TO_USINT(SHR(Axis.DrvToPlc.CfgValueIn,8));
			TextStringletsBA[18]:= UDINT_TO_USINT(SHR(Axis.DrvToPlc.CfgValueIn,16));
			TextStringletsBA[19]:= UDINT_TO_USINT(SHR(Axis.DrvToPlc.CfgValueIn,24));
			uiState := 7;
		END_IF

	(*Get Stringlet 5*)
	7:	Axis.PlcToDrv.CfgControlWord := 16#7406;
		Axis.PlcToDrv.CfgIndexOut := ErrorCode;
		Axis.PlcToDrv.CfgValueOut := 5; (*Stringlet 5*)
		fTimer(IN:=TRUE,PT:=tiT1);

		IF fTimer.Q THEN
			fTimer(IN:=FALSE);
			ErrorID := 16#01; (*fTimer error: No response from drive*)
			uiState := 90;
		END_IF

		IF Axis.DrvToPlc.CfgStatusWord = 16#0006 THEN
			fTimer(IN:=FALSE);
			TextStringletsBA[20]:= UDINT_TO_USINT(Axis.DrvToPlc.CfgValueIn);
			TextStringletsBA[21]:= UDINT_TO_USINT(SHR(Axis.DrvToPlc.CfgValueIn,8));
			TextStringletsBA[22]:= UDINT_TO_USINT(SHR(Axis.DrvToPlc.CfgValueIn,16));
			TextStringletsBA[23]:= UDINT_TO_USINT(SHR(Axis.DrvToPlc.CfgValueIn,24));
			uiState := 8;
		END_IF

	(*Get Stringlet 6*)
	8:	Axis.PlcToDrv.CfgControlWord := 16#7407;
		Axis.PlcToDrv.CfgIndexOut := ErrorCode;
		Axis.PlcToDrv.CfgValueOut := 6; (*Stringlet 6*)
		fTimer(IN:=TRUE,PT:=tiT1);

		IF fTimer.Q THEN
			fTimer(IN:=FALSE);
			ErrorID := 16#01; (*fTimer error: No response from drive*)
			uiState := 90;
		END_IF

		IF Axis.DrvToPlc.CfgStatusWord = 16#0007 THEN
			fTimer(IN:=FALSE);
			TextStringletsBA[24]:= UDINT_TO_USINT(Axis.DrvToPlc.CfgValueIn);
			TextStringletsBA[25]:= UDINT_TO_USINT(SHR(Axis.DrvToPlc.CfgValueIn,8));
			TextStringletsBA[26]:= UDINT_TO_USINT(SHR(Axis.DrvToPlc.CfgValueIn,16));
			TextStringletsBA[27]:= UDINT_TO_USINT(SHR(Axis.DrvToPlc.CfgValueIn,24));
			uiState := 9;
		END_IF

	(*Get Stringlet 7*)
	9:	Axis.PlcToDrv.CfgControlWord := 16#7408;
		Axis.PlcToDrv.CfgIndexOut := ErrorCode;
		Axis.PlcToDrv.CfgValueOut := 7; (*Stringlet 7*)
		fTimer(IN:=TRUE,PT:=tiT1);

		IF fTimer.Q THEN
			fTimer(IN:=FALSE);
			ErrorID := 16#01; (*fTimer error: No response from drive*)
			uiState := 90;
		END_IF

		IF Axis.DrvToPlc.CfgStatusWord = 16#0008 THEN
			fTimer(IN:=FALSE);
			TextStringletsBA[28]:= UDINT_TO_USINT(Axis.DrvToPlc.CfgValueIn);
			TextStringletsBA[29]:= UDINT_TO_USINT(SHR(Axis.DrvToPlc.CfgValueIn,8));
			TextStringletsBA[30]:= UDINT_TO_USINT(SHR(Axis.DrvToPlc.CfgValueIn,16));
			TextStringletsBA[31]:= UDINT_TO_USINT(SHR(Axis.DrvToPlc.CfgValueIn,24));
			ErrorText := '';
			FOR i := 0 TO 31 DO
				TextStringletsS[i] := USINT_TO_ASCIISTRING(TextStringletsBA[i]);
				ErrorText := CONCAT(ErrorText, TextStringletsS[i]);
			END_FOR
			uiState := 100;
		END_IF

(*=============================================================================
*  Error State
===============================================================================*)    

	(*Error State I*)
	90:	IF Busy THEN
			Axis.ConfigChannelBusy := FALSE; (*Only reset ConfigChannelBusy if function block is Busy*)
			Axis.PlcToDrv.CfgControlWord := 16#0000; (*Reset Config Control*)
		END_IF

		Error := TRUE;
		Busy := FALSE;
		Done := FALSE;
		ErrorText := '';
		fTimer(IN:=FALSE);
		i := 0;

		uiState := 91;

	(*Error State II*)
	91:	IF NOT Execute THEN
			Error := FALSE;
			ErrorID := 0;
			uiState := 0;
		END_IF

(*=============================================================================
*  Command Done
===============================================================================*)    

	(*Command succesfully executed*)
	100:Done := TRUE;
		Busy := FALSE;
		fTimer(IN:=FALSE);
		i := 0;

		Axis.ConfigChannelBusy := FALSE;
		Axis.PlcToDrv.CfgControlWord := 16#0000; (*Reset Config Control*)

		uiState := 101;

	(*Wait Not Execute*)
	101:IF NOT Execute THEN
			Done := FALSE;
			ErrorText := '';
			uiState := 0;
		END_IF

END_CASE

END_FUNCTION_BLOCK

// POUs/LinMot Functions/USINT_TO_ASCIISTRING
FUNCTION USINT_TO_ASCIISTRING : STRING(1)
VAR_INPUT
	Value	:USINT;
END_VAR
VAR
	str1	:STRING(1);
	pstr	:POINTER TO BYTE;
	digit	:BYTE;
END_VAR
(*Version history:
Date         	 | Version    		| Created under     	| Author          	| Remark 
------------------------------------------------------------------------------------------------------------------------------- 
2012-oct-12   	 | 1.0.0      		| V2.11.0 (Build 1016)	| fj  				| initial release with pointer
*)

(*This function returns a character based on the input value*)
str1 := '@';
pstr := ADR(str1);
digit :=USINT_TO_BYTE(Value);
pstr^ := digit;
USINT_TO_ASCIISTRING := str1;

END_FUNCTION

